C05448=1100.814,341.795,-85.952,179.336,18.021,152.003
C05449=1100.819,342.043,-85.985,179.340,18.025,152.003
C05450=1100.825,342.291,-86.018,179.342,18.028,152.003
C05451=1100.831,342.538,-86.052,179.345,18.031,152.004
C05452=1100.839,342.910,-86.102,179.350,18.036,152.004
C05453=1100.848,343.283,-86.153,179.355,18.040,152.004
C05454=1100.856,343.656,-86.204,179.360,18.045,152.004
C05455=1100.865,344.027,-86.255,179.364,18.049,152.004
C05456=1100.870,344.275,-86.288,179.368,18.053,152.005
C05457=1100.876,344.523,-86.321,179.371,18.056,152.005
C05458=1100.882,344.770,-86.355,179.374,18.059,152.005
C05459=1100.887,345.018,-86.389,179.377,18.062,152.005
C05460=1100.893,345.265,-86.423,179.380,18.065,152.005
C05461=1100.899,345.514,-86.456,179.384,18.069,152.005
C05462=1100.905,345.761,-86.490,179.386,18.072,152.006
C05463=1100.911,346.009,-86.524,179.389,18.075,152.006
C05464=1100.916,346.256,-86.558,179.393,18.078,152.006
C05465=1100.922,346.503,-86.592,179.395,18.082,152.006
C05466=1100.927,346.752,-86.626,179.399,18.085,152.006
C05467=1100.933,346.999,-86.660,179.402,18.088,152.006
C05468=1100.939,347.247,-86.693,179.405,18.091,152.007
C05469=1100.944,347.494,-86.727,179.408,18.095,152.007
C05470=1100.950,347.741,-86.761,179.411,18.098,152.007
C05471=1100.956,347.989,-86.795,179.415,18.101,152.007
C05472=1100.961,348.237,-86.829,179.417,18.104,152.008
C05473=1100.967,348.485,-86.864,179.421,18.108,152.008
C05474=1100.973,348.733,-86.897,179.424,18.111,152.008
C05475=1100.979,348.980,-86.931,179.426,18.114,152.008
C05476=1100.985,349.227,-86.965,179.430,18.118,152.008
C05477=1100.990,349.475,-87.000,179.433,18.121,152.009
C05478=1100.995,349.723,-87.033,179.436,18.125,152.009
C05479=1101.001,349.970,-87.067,179.439,18.128,152.009
C05480=1101.008,350.218,-87.102,179.443,18.132,152.009
C05481=1101.013,350.466,-87.136,179.445,18.135,152.010
C05482=1101.019,350.713,-87.170,179.449,18.138,152.010
C05483=1101.024,350.961,-87.204,179.452,18.142,152.010
C05484=1101.029,351.209,-87.238,179.454,18.145,152.010
C05485=1101.035,351.456,-87.272,179.458,18.149,152.010
C05486=1101.042,351.704,-87.307,179.461,18.151,152.011
C05487=1101.047,351.951,-87.341,179.464,18.155,152.011
C05488=1101.053,352.199,-87.375,179.467,18.159,152.011
C05489=1101.059,352.446,-87.410,179.470,18.162,152.011
C05490=1101.064,352.694,-87.445,179.473,18.166,152.012
C05491=1101.070,352.942,-87.479,179.477,18.169,152.012
C05492=1101.076,353.189,-87.513,179.479,18.172,152.012
C05493=1101.081,353.436,-87.547,179.483,18.176,152.012
C05494=1101.087,353.684,-87.581,179.485,18.179,152.013
C05495=1101.093,353.932,-87.616,179.489,18.183,152.013
C05496=1101.099,354.179,-87.650,179.491,18.187,152.013
C05497=1101.104,354.427,-87.684,179.495,18.190,152.014
C05498=1101.109,354.674,-87.719,179.497,18.194,152.014
C05499=1101.116,354.922,-87.754,179.501,18.197,152.014
C05500=1101.121,355.170,-87.788,179.504,18.201,152.014
C05501=1101.127,355.417,-87.822,179.507,18.205,152.015
C05502=1101.132,355.664,-87.858,179.509,18.208,152.015
C05503=1101.139,355.912,-87.892,179.513,18.212,152.015
C05504=1101.147,356.286,-87.944,179.518,18.218,152.016
C05505=1101.156,356.660,-87.996,179.522,18.223,152.016
C05506=1101.164,357.035,-88.049,179.526,18.228,152.017
C05507=1101.172,357.410,-88.101,179.531,18.234,152.017
C05508=1101.179,357.657,-88.137,179.534,18.238,152.017
C05509=1101.184,357.905,-88.171,179.537,18.241,152.018
C05510=1101.190,358.152,-88.205,179.540,18.245,152.018
C05511=1101.196,358.400,-88.241,179.544,18.249,152.018
C05512=1101.202,358.647,-88.275,179.546,18.253,152.019
C05513=1101.207,358.895,-88.310,179.550,18.256,152.019
C05514=1101.213,359.143,-88.345,179.552,18.260,152.019
C05515=1101.219,359.390,-88.379,179.555,18.264,152.020
C05516=1101.224,359.637,-88.414,179.558,18.267,152.020
C05517=1101.231,359.885,-88.449,179.561,18.271,152.021
C05518=1101.236,360.132,-88.484,179.565,18.275,152.021
C05519=1101.241,360.379,-88.519,179.567,18.279,152.021
C05520=1101.248,360.627,-88.554,179.571,18.283,152.022
C05521=1101.253,360.874,-88.589,179.573,18.286,152.022
C05522=1101.258,361.122,-88.624,179.576,18.290,152.022
C05523=1101.264,361.370,-88.659,179.580,18.295,152.023
C05524=1101.270,361.617,-88.693,179.582,18.298,152.023
C05525=1101.276,361.865,-88.729,179.585,18.302,152.023
C05526=1101.281,362.112,-88.764,179.588,18.306,152.024
C05527=1101.287,362.359,-88.799,179.591,18.310,152.024
C05528=1101.293,362.606,-88.834,179.594,18.314,152.025
C05529=1101.299,362.854,-88.869,179.597,18.317,152.025
C05530=1101.305,363.102,-88.905,179.600,18.322,152.025
C05531=1101.310,363.349,-88.939,179.602,18.325,152.026
C05532=1101.316,363.597,-88.975,179.606,18.329,152.026
C05533=1101.322,363.844,-89.010,179.609,18.333,152.027
C05534=1101.327,364.091,-89.045,179.611,18.337,152.027
C05535=1101.333,364.339,-89.080,179.615,18.341,152.027
C05536=1101.339,364.586,-89.116,179.618,18.346,152.028
C05537=1101.345,364.834,-89.151,179.620,18.349,152.028
C05538=1101.350,365.081,-89.186,179.623,18.353,152.029
C05539=1101.356,365.329,-89.221,179.627,18.358,152.029
C05540=1101.362,365.575,-89.256,179.629,18.361,152.030
C05541=1101.368,365.823,-89.292,179.632,18.366,152.030
C05542=1101.373,366.070,-89.328,179.635,18.370,152.030
C05543=1101.379,366.318,-89.363,179.638,18.374,152.031
C05544=1101.384,366.565,-89.398,179.641,18.378,152.031
C05545=1101.390,366.812,-89.433,179.644,18.382,152.032
C05546=1101.396,367.060,-89.469,179.647,18.386,152.032
C05547=1101.401,367.307,-89.504,179.650,18.390,152.033
C05548=1101.407,367.555,-89.540,179.653,18.395,152.033
C05549=1101.413,367.802,-89.576,179.656,18.399,152.034
C05550=1101.419,368.049,-89.611,179.658,18.403,152.034
C05551=1101.424,368.296,-89.647,179.661,18.407,152.035
C05552=1101.430,368.544,-89.682,179.665,18.411,152.035
C05553=1101.436,368.791,-89.718,179.667,18.415,152.036
C05554=1101.442,369.039,-89.753,179.670,18.420,152.036
C05555=1101.446,369.286,-89.789,179.673,18.424,152.037
C05556=1101.456,369.675,-89.845,179.677,18.431,152.037
C05557=1101.465,370.065,-89.902,179.682,18.438,152.038
C05558=1101.474,370.455,-89.957,179.686,18.444,152.039
C05559=1101.483,370.844,-90.013,179.691,18.451,152.040
C05560=1101.489,371.092,-90.049,179.693,18.455,152.040
C05561=1101.494,371.339,-90.085,179.697,18.459,152.041
C05562=1101.500,371.586,-90.122,179.700,18.464,152.041
C05563=1101.506,371.833,-90.157,179.703,18.469,152.042
C05564=1101.512,372.081,-90.193,179.705,18.472,152.042
C05565=1101.518,372.328,-90.228,179.708,18.477,152.043
C05566=1101.523,372.575,-90.264,179.711,18.482,152.043
C05567=1101.530,372.822,-90.300,179.714,18.486,152.044
C05568=1101.534,373.069,-90.336,179.717,18.491,152.045
C05569=1101.540,373.317,-90.372,179.719,18.495,152.045
C05570=1101.547,373.564,-90.408,179.722,18.499,152.046
C05571=1101.552,373.811,-90.444,179.725,18.503,152.046
C05572=1101.558,374.059,-90.479,179.728,18.508,152.047
C05573=1101.564,374.306,-90.516,179.730,18.512,152.047
C05574=1101.569,374.553,-90.552,179.733,18.517,152.048
C05575=1101.575,374.800,-90.588,179.736,18.521,152.048
C05576=1101.581,375.048,-90.625,179.739,18.526,152.049
C05577=1101.586,375.295,-90.660,179.742,18.531,152.050
C05578=1101.592,375.542,-90.696,179.745,18.535,152.050
C05579=1101.597,375.790,-90.732,179.747,18.540,152.051
C05580=1101.603,376.037,-90.769,179.750,18.545,152.052
C05581=1101.610,376.284,-90.805,179.753,18.549,152.052
C05582=1101.615,376.531,-90.841,179.756,18.554,152.053
C05583=1101.621,376.779,-90.877,179.759,18.559,152.053
C05584=1101.626,377.026,-90.914,179.762,18.564,152.054
C05585=1101.632,377.273,-90.949,179.765,18.568,152.055
C05586=1101.638,377.520,-90.986,179.767,18.572,152.055
C05587=1101.643,377.767,-91.023,179.769,18.577,152.056
C05588=1101.649,378.014,-91.058,179.772,18.582,152.057
C05589=1101.655,378.262,-91.095,179.775,18.587,152.057
C05590=1101.661,378.509,-91.131,179.778,18.592,152.058
C05591=1101.666,378.757,-91.168,179.781,18.596,152.058
C05592=1101.672,379.003,-91.204,179.784,18.601,152.059
C05593=1101.677,379.251,-91.240,179.787,18.606,152.060
C05594=1101.684,379.498,-91.277,179.789,18.610,152.060
C05595=1101.689,379.746,-91.314,179.792,18.615,152.061
C05596=1101.695,379.992,-91.350,179.794,18.620,152.062
C05597=1101.700,380.240,-91.386,179.797,18.625,152.062
C05598=1101.706,380.487,-91.423,179.800,18.630,152.063
C05599=1101.712,380.734,-91.460,179.803,18.635,152.064
C05600=1101.718,380.981,-91.496,179.806,18.640,152.064
C05601=1101.723,381.228,-91.533,179.808,18.645,152.065
C05602=1101.729,381.476,-91.569,179.811,18.650,152.066
C05603=1101.735,381.723,-91.606,179.814,18.655,152.067
C05604=1101.741,381.970,-91.642,179.817,18.659,152.067
C05605=1101.746,382.217,-91.679,179.819,18.664,152.068
C05606=1101.753,382.464,-91.715,179.822,18.669,152.069
C05607=1101.758,382.711,-91.752,179.824,18.674,152.069
C05608=1101.768,383.128,-91.814,179.829,18.683,152.071
C05609=1101.777,383.543,-91.876,179.833,18.691,152.072
C05610=1101.787,383.960,-91.938,179.838,18.700,152.073
C05611=1101.796,384.376,-92.000,179.843,18.708,152.074
C05612=1101.802,384.624,-92.037,179.845,18.714,152.075
C05613=1101.808,384.871,-92.073,179.848,18.719,152.076
C05614=1101.814,385.118,-92.111,179.850,18.724,152.077
C05615=1101.820,385.366,-92.148,179.853,18.729,152.078
C05616=1101.825,385.612,-92.185,179.856,18.734,152.078
C05617=1101.831,385.859,-92.221,179.858,18.739,152.079
C05618=1101.837,386.106,-92.258,179.861,18.745,152.080
C05619=1101.842,386.353,-92.295,179.864,18.750,152.081
C05620=1101.848,386.601,-92.333,179.866,18.755,152.082
C05621=1101.854,386.848,-92.370,179.869,18.760,152.082
C05622=1101.860,387.095,-92.407,179.871,18.766,152.083
C05623=1101.865,387.341,-92.443,179.874,18.771,152.084
C05624=1101.871,387.589,-92.480,179.877,18.777,152.085
C05625=1101.876,387.836,-92.517,179.880,18.782,152.086
C05626=1101.882,388.083,-92.555,179.882,18.787,152.087
C05627=1101.888,388.330,-92.592,179.885,18.793,152.087
C05628=1101.894,388.577,-92.629,179.888,18.798,152.088
C05629=1101.900,388.824,-92.666,179.890,18.803,152.089
C05630=1101.906,389.071,-92.703,179.893,18.809,152.090
C05631=1101.911,389.319,-92.741,179.895,18.814,152.091
C05632=1101.917,389.565,-92.778,179.898,18.820,152.092
C05633=1101.923,389.813,-92.815,179.900,18.825,152.092
C05634=1101.929,390.059,-92.853,179.903,18.830,152.093
C05635=1101.934,390.307,-92.890,179.906,18.836,152.094
C05636=1101.940,390.554,-92.928,179.909,18.842,152.095
C05637=1101.947,390.801,-92.964,179.911,18.847,152.096
C05638=1101.953,391.047,-93.002,179.913,18.852,152.097
C05639=1101.958,391.295,-93.039,179.916,18.858,152.098
C05640=1101.964,391.541,-93.077,179.918,18.863,152.099
C05641=1101.970,391.789,-93.114,179.921,18.869,152.100
C05642=1101.976,392.036,-93.152,179.923,18.875,152.101
C05643=1101.981,392.283,-93.189,179.926,18.881,152.101
C05644=1101.987,392.530,-93.226,179.929,18.886,152.102
C05645=1101.993,392.777,-93.264,179.931,18.892,152.103
C05646=1101.999,393.024,-93.301,179.934,18.897,152.104
C05647=1102.004,393.271,-93.340,179.936,18.903,152.105
C05648=1102.009,393.518,-93.377,179.938,18.909,152.106
C05649=1102.015,393.765,-93.414,179.942,18.915,152.107
C05650=1102.021,394.012,-93.452,179.944,18.921,152.108
C05651=1102.027,394.259,-93.489,179.946,18.926,152.109
C05652=1102.033,394.507,-93.527,179.949,18.932,152.110
C05653=1102.039,394.753,-93.565,179.951,18.938,152.111
C05654=1102.044,395.000,-93.603,179.953,18.943,152.112
C05655=1102.050,395.248,-93.640,179.956,18.950,152.113
C05656=1102.056,395.494,-93.678,179.959,18.955,152.114
C05657=1102.062,395.741,-93.716,179.961,18.961,152.115
C05658=1102.068,395.988,-93.754,179.963,18.967,152.116
C05659=1102.072,396.236,-93.791,179.966,18.973,152.117
C05660=1102.078,396.450,-93.824,179.968,18.978,152.118
C05661=1102.083,396.665,-93.857,179.970,18.984,152.119
C05662=1102.088,396.878,-93.890,179.972,18.989,152.120
C05663=1102.093,397.093,-93.924,179.975,18.994,152.121
C05664=1102.098,397.307,-93.955,179.976,18.999,152.121
C05665=1102.103,397.521,-93.989,179.979,19.004,152.122
C05666=1102.108,397.737,-94.022,179.980,19.010,152.123
C05667=1102.113,397.950,-94.055,179.983,19.015,152.124
C05668=1102.118,398.197,-94.093,179.985,19.021,152.125
C05669=1102.125,398.445,-94.131,179.988,19.027,152.126
C05670=1102.131,398.691,-94.169,179.990,19.033,152.128
C05671=1102.136,398.938,-94.207,179.992,19.039,152.129
C05672=1102.142,399.185,-94.245,179.995,19.045,152.130
C05673=1102.148,399.432,-94.283,179.998,19.052,152.131
C05674=1102.153,399.680,-94.321,180.000,19.058,152.132
C05675=1102.159,399.926,-94.359,-179.998,19.064,152.133
C05676=1102.164,400.173,-94.398,-179.995,19.070,152.134
C05677=1102.171,400.421,-94.436,-179.993,19.077,152.135
C05678=1102.176,400.668,-94.474,-179.991,19.083,152.136
C05679=1102.182,400.915,-94.512,-179.988,19.089,152.137
C05680=1102.188,401.161,-94.550,-179.986,19.096,152.139
C05681=1102.194,401.408,-94.589,-179.984,19.102,152.140
C05682=1102.199,401.656,-94.627,-179.981,19.109,152.141
C05683=1102.205,401.902,-94.665,-179.979,19.115,152.142
C05684=1102.210,402.149,-94.703,-179.976,19.122,152.143
C05685=1102.217,402.396,-94.742,-179.974,19.128,152.144
C05686=1102.222,402.643,-94.781,-179.972,19.134,152.146
C05687=1102.228,402.890,-94.818,-179.969,19.141,152.147
C05688=1102.234,403.138,-94.857,-179.967,19.147,152.148
C05689=1102.240,403.384,-94.896,-179.964,19.154,152.149
C05690=1102.245,403.631,-94.934,-179.962,19.160,152.150
C05691=1102.252,403.878,-94.972,-179.960,19.167,152.152
C05692=1102.257,404.125,-95.011,-179.958,19.173,152.153
C05693=1102.262,404.372,-95.049,-179.956,19.180,152.154
C05694=1102.269,404.619,-95.088,-179.953,19.187,152.155
C05695=1102.274,404.866,-95.127,-179.951,19.193,152.156
C05696=1102.279,405.113,-95.165,-179.948,19.200,152.158
C05697=1102.286,405.360,-95.204,-179.946,19.206,152.159
C05698=1102.291,405.607,-95.242,-179.944,19.214,152.160
C05699=1102.297,405.854,-95.282,-179.942,19.220,152.162
C05700=1102.303,406.101,-95.319,-179.939,19.227,152.163
C05701=1102.309,406.347,-95.358,-179.937,19.234,152.164
C05702=1102.315,406.595,-95.397,-179.935,19.241,152.165
C05703=1102.320,406.841,-95.436,-179.932,19.247,152.167
C05704=1102.327,407.089,-95.474,-179.930,19.254,152.168
C05705=1102.332,407.335,-95.513,-179.927,19.262,152.169
C05706=1102.337,407.582,-95.552,-179.925,19.268,152.171
C05707=1102.343,407.829,-95.591,-179.923,19.275,152.172
C05708=1102.349,408.076,-95.630,-179.921,19.282,152.173
C05709=1102.355,408.323,-95.668,-179.918,19.289,152.175
C05710=1102.361,408.570,-95.707,-179.917,19.296,152.176
C05711=1102.367,408.817,-95.747,-179.914,19.303,152.177
C05712=1102.372,409.064,-95.785,-179.912,19.311,152.179
C05713=1102.377,409.310,-95.824,-179.910,19.317,152.180
C05714=1102.384,409.557,-95.864,-179.907,19.325,152.181
C05715=1102.389,409.804,-95.903,-179.905,19.332,152.183
C05716=1102.394,410.018,-95.936,-179.903,19.338,152.184
C05717=1102.399,410.233,-95.970,-179.902,19.344,152.185
C05718=1102.404,410.447,-96.004,-179.900,19.351,152.186
C05719=1102.409,410.661,-96.038,-179.898,19.357,152.188
C05720=1102.414,410.876,-96.072,-179.896,19.363,152.189
C05721=1102.419,411.090,-96.106,-179.894,19.370,152.190
C05722=1102.424,411.304,-96.140,-179.892,19.376,152.191
C05723=1102.429,411.519,-96.174,-179.890,19.382,152.193
C05724=1102.435,411.766,-96.213,-179.887,19.390,152.194
C05725=1102.441,412.012,-96.252,-179.886,19.397,152.196
C05726=1102.447,412.259,-96.292,-179.883,19.405,152.197
C05727=1102.452,412.506,-96.331,-179.881,19.412,152.198
C05728=1102.458,412.753,-96.370,-179.878,19.419,152.200
C05729=1102.464,412.999,-96.409,-179.877,19.426,152.201
C05730=1102.470,413.247,-96.449,-179.874,19.434,152.203
C05731=1102.476,413.494,-96.488,-179.872,19.442,152.204
C05732=1102.481,413.740,-96.527,-179.870,19.450,152.206
C05733=1102.487,413.988,-96.567,-179.868,19.457,152.207
C05734=1102.492,414.234,-96.606,-179.866,19.464,152.209
C05735=1102.498,414.481,-96.646,-179.863,19.472,152.210
C05736=1102.505,414.728,-96.686,-179.861,19.480,152.212
C05737=1102.510,414.974,-96.725,-179.859,19.487,152.213
C05738=1102.516,415.221,-96.764,-179.857,19.495,152.215
C05739=1102.522,415.468,-96.803,-179.855,19.502,152.216
C05740=1102.528,415.715,-96.843,-179.853,19.510,152.218
C05741=1102.534,415.961,-96.883,-179.850,19.518,152.220
C05742=1102.540,416.208,-96.922,-179.848,19.526,152.221
C05743=1102.546,416.455,-96.961,-179.846,19.534,152.223
C05744=1102.551,416.702,-97.001,-179.844,19.541,152.224
C05745=1102.557,416.948,-97.041,-179.842,19.549,152.226
C05746=1102.563,417.195,-97.081,-179.840,19.557,152.227
C05747=1102.569,417.442,-97.120,-179.838,19.565,152.229
C05748=1102.574,417.689,-97.160,-179.836,19.573,152.231
C05749=1102.580,417.936,-97.200,-179.833,19.581,152.232
C05750=1102.586,418.183,-97.239,-179.831,19.590,152.234
C05751=1102.591,418.429,-97.280,-179.829,19.598,152.236
C05752=1102.597,418.676,-97.319,-179.827,19.606,152.237
C05753=1102.603,418.922,-97.359,-179.825,19.614,152.239
C05754=1102.608,419.169,-97.399,-179.823,19.622,152.241
C05755=1102.615,419.416,-97.439,-179.821,19.630,152.242
C05756=1102.621,419.663,-97.478,-179.819,19.638,152.244
C05757=1102.626,419.909,-97.519,-179.817,19.647,152.246
C05758=1102.632,420.156,-97.558,-179.815,19.655,152.247
C05759=1102.638,420.403,-97.598,-179.813,19.664,152.249
C05760=1102.643,420.649,-97.639,-179.810,19.671,152.251
C05761=1102.649,420.896,-97.678,-179.808,19.680,152.253
C05762=1102.655,421.143,-97.719,-179.806,19.688,152.254
C05763=1102.661,421.390,-97.758,-179.804,19.697,152.256
C05764=1102.667,421.636,-97.798,-179.802,19.705,152.258
C05765=1102.673,421.883,-97.839,-179.800,19.713,152.260
C05766=1102.679,422.129,-97.879,-179.799,19.722,152.261
C05767=1102.684,422.377,-97.919,-179.797,19.731,152.263
C05768=1102.691,422.623,-97.959,-179.795,19.739,152.265
C05769=1102.696,422.869,-98.000,-179.793,19.747,152.267
C05770=1102.702,423.116,-98.040,-179.791,19.756,152.269
C05771=1102.707,423.363,-98.080,-179.789,19.764,152.270
C05772=1102.713,423.584,-98.116,-179.787,19.773,152.272
C05773=1102.718,423.805,-98.152,-179.785,19.780,152.274
C05774=1102.723,424.026,-98.189,-179.783,19.789,152.275
C05775=1102.728,424.248,-98.225,-179.782,19.796,152.277
C05776=1102.733,424.468,-98.260,-179.780,19.804,152.279
C05777=1102.738,424.689,-98.297,-179.778,19.812,152.280
C05778=1102.744,424.910,-98.333,-179.776,19.820,152.282
C05779=1102.749,425.132,-98.369,-179.775,19.828,152.284
C05780=1102.755,425.378,-98.409,-179.772,19.837,152.286
C05781=1102.760,425.625,-98.450,-179.771,19.846,152.288
C05782=1102.766,425.871,-98.491,-179.769,19.855,152.290
C05783=1102.772,426.118,-98.531,-179.767,19.863,152.291
C05784=1102.778,426.365,-98.571,-179.765,19.873,152.294
C05785=1102.784,426.611,-98.613,-179.763,19.882,152.295
C05786=1102.790,426.857,-98.653,-179.761,19.891,152.297
C05787=1102.795,427.104,-98.693,-179.759,19.900,152.299
C05788=1102.801,427.350,-98.734,-179.758,19.909,152.301
C05789=1102.807,427.597,-98.774,-179.755,19.919,152.303
C05790=1102.813,427.844,-98.815,-179.754,19.927,152.305
C05791=1102.819,428.091,-98.856,-179.752,19.937,152.307
C05792=1102.825,428.337,-98.897,-179.750,19.946,152.309
C05793=1102.831,428.583,-98.937,-179.748,19.956,152.311
C05794=1102.837,428.830,-98.978,-179.746,19.965,152.313
C05795=1102.842,429.077,-99.019,-179.745,19.974,152.315
C05796=1102.848,429.322,-99.060,-179.742,19.984,152.317
C05797=1102.854,429.569,-99.100,-179.741,19.993,152.320
C05798=1102.860,429.816,-99.141,-179.739,20.002,152.322
C05799=1102.866,430.062,-99.182,-179.737,20.012,152.324
C05800=1102.871,430.309,-99.223,-179.735,20.022,152.326
C05801=1102.877,430.555,-99.265,-179.734,20.031,152.328
C05802=1102.883,430.802,-99.305,-179.732,20.041,152.330
C05803=1102.889,431.049,-99.346,-179.730,20.050,152.332
C05804=1102.894,431.295,-99.388,-179.729,20.060,152.334
C05805=1102.900,431.542,-99.428,-179.727,20.070,152.337
C05806=1102.906,431.788,-99.470,-179.725,20.080,152.339
C05807=1102.912,432.035,-99.510,-179.723,20.090,152.341
C05808=1102.918,432.281,-99.551,-179.722,20.099,152.343
C05809=1102.924,432.527,-99.593,-179.720,20.109,152.345
C05810=1102.930,432.774,-99.634,-179.718,20.119,152.348
C05811=1102.936,433.020,-99.675,-179.717,20.129,152.350
C05812=1102.942,433.267,-99.716,-179.715,20.139,152.352
C05813=1102.948,433.513,-99.757,-179.713,20.149,152.354
C05814=1102.953,433.759,-99.799,-179.711,20.159,152.356
C05815=1102.958,434.006,-99.840,-179.710,20.169,152.359
C05816=1102.964,434.252,-99.881,-179.708,20.180,152.361
C05817=1102.970,434.499,-99.923,-179.707,20.190,152.363
C05818=1102.976,434.745,-99.964,-179.705,20.200,152.366
C05819=1102.982,434.992,-100.005,-179.703,20.210,152.368
C05820=1102.988,435.238,-100.047,-179.701,20.221,152.370
C05821=1102.994,435.484,-100.088,-179.700,20.231,152.373
C05822=1102.999,435.731,-100.130,-179.698,20.242,152.375
C05823=1103.005,435.977,-100.172,-179.697,20.251,152.377
C05824=1103.011,436.223,-100.213,-179.695,20.262,152.380
C05825=1103.017,436.469,-100.254,-179.694,20.272,152.382
C05826=1103.022,436.716,-100.295,-179.692,20.283,152.385
C05827=1103.028,436.963,-100.337,-179.690,20.294,152.387
C05828=1103.038,437.358,-100.404,-179.688,20.311,152.391
C05829=1103.047,437.753,-100.471,-179.685,20.328,152.395
C05830=1103.056,438.149,-100.538,-179.684,20.345,152.399
C05831=1103.066,438.544,-100.605,-179.681,20.362,152.403
C05832=1103.072,438.791,-100.647,-179.679,20.374,152.405
C05833=1103.077,439.037,-100.688,-179.678,20.384,152.408
C05834=1103.083,439.283,-100.730,-179.676,20.395,152.410
C05835=1103.089,439.530,-100.772,-179.674,20.406,152.413
C05836=1103.095,439.776,-100.814,-179.674,20.417,152.415
C05837=1103.101,440.022,-100.856,-179.672,20.428,152.418
C05838=1103.107,440.268,-100.897,-179.670,20.439,152.420
C05839=1103.113,440.515,-100.939,-179.669,20.450,152.423
C05840=1103.119,440.761,-100.981,-179.668,20.461,152.426
C05841=1103.125,441.008,-101.024,-179.666,20.473,152.428
C05842=1103.131,441.254,-101.065,-179.664,20.484,152.431
C05843=1103.136,441.500,-101.108,-179.664,20.495,152.433
C05844=1103.142,441.746,-101.150,-179.662,20.507,152.436
C05845=1103.148,441.992,-101.191,-179.661,20.518,152.439
C05846=1103.154,442.239,-101.234,-179.659,20.530,152.442
C05847=1103.160,442.485,-101.276,-179.657,20.541,152.444
C05848=1103.165,442.731,-101.318,-179.657,20.552,152.447
C05849=1103.172,442.977,-101.360,-179.655,20.564,152.450
C05850=1103.177,443.223,-101.402,-179.654,20.576,152.453
C05851=1103.183,443.470,-101.445,-179.652,20.588,152.455
C05852=1103.189,443.716,-101.487,-179.652,20.599,152.458
C05853=1103.194,443.962,-101.529,-179.650,20.611,152.461
C05854=1103.201,444.208,-101.572,-179.650,20.622,152.464
C05855=1103.206,444.455,-101.614,-179.649,20.635,152.466
C05856=1103.212,444.701,-101.657,-179.648,20.646,152.469
C05857=1103.218,444.947,-101.698,-179.648,20.658,152.472
C05858=1103.224,445.194,-101.741,-179.647,20.669,152.475
C05859=1103.230,445.439,-101.784,-179.648,20.680,152.478
C05860=1103.235,445.686,-101.826,-179.647,20.692,152.481
C05861=1103.242,445.932,-101.869,-179.648,20.703,152.484
C05862=1103.248,446.178,-101.911,-179.647,20.715,152.487
C05863=1103.253,446.424,-101.953,-179.648,20.727,152.490
C05864=1103.259,446.671,-101.996,-179.648,20.738,152.493
C05865=1103.265,446.917,-102.039,-179.649,20.749,152.496
C05866=1103.270,447.163,-102.082,-179.650,20.761,152.499
C05867=1103.277,447.410,-102.123,-179.650,20.772,152.502
C05868=1103.282,447.656,-102.166,-179.651,20.784,152.505
C05869=1103.288,447.901,-102.209,-179.652,20.795,152.508
C05870=1103.294,448.148,-102.252,-179.653,20.807,152.511
C05871=1103.300,448.394,-102.294,-179.654,20.818,152.514
C05872=1103.306,448.641,-102.337,-179.655,20.830,152.517
C05873=1103.312,448.887,-102.379,-179.657,20.841,152.521
C05874=1103.317,449.133,-102.422,-179.658,20.852,152.524
C05875=1103.323,449.379,-102.465,-179.660,20.864,152.527
C05876=1103.329,449.625,-102.508,-179.662,20.875,152.530
C05877=1103.336,449.871,-102.551,-179.663,20.886,152.533
C05878=1103.341,450.117,-102.593,-179.665,20.898,152.536
C05879=1103.347,450.364,-102.637,-179.667,20.909,152.539
C05880=1102.945,450.357,-102.771,-179.739,21.135,152.609
C05881=1102.939,450.111,-102.728,-179.737,21.124,152.606
C05882=1102.933,449.864,-102.685,-179.736,21.112,152.603
C05883=1102.928,449.618,-102.642,-179.734,21.101,152.599
C05884=1102.921,449.372,-102.600,-179.732,21.090,152.596
C05885=1102.915,449.126,-102.557,-179.731,21.078,152.593
C05886=1102.910,448.880,-102.514,-179.729,21.067,152.590
C05887=1102.904,448.633,-102.471,-179.728,21.055,152.587
C05888=1102.898,448.388,-102.428,-179.727,21.044,152.584
C05889=1102.892,448.141,-102.385,-179.725,21.033,152.581
C05890=1102.886,447.895,-102.343,-179.725,21.021,152.577
C05891=1102.880,447.648,-102.301,-179.723,21.010,152.574
C05892=1102.874,447.402,-102.258,-179.723,20.998,152.571
C05893=1102.869,447.156,-102.215,-179.722,20.986,152.568
C05894=1102.863,446.910,-102.172,-179.722,20.974,152.565
C05895=1102.857,446.664,-102.130,-179.721,20.963,152.562
C05896=1102.851,446.418,-102.087,-179.721,20.951,152.559
C05897=1102.845,446.171,-102.045,-179.720,20.940,152.556
C05898=1102.840,445.925,-102.002,-179.721,20.928,152.553
C05899=1102.833,445.679,-101.959,-179.720,20.917,152.550
C05900=1102.827,445.433,-101.916,-179.721,20.905,152.547
C05901=1102.822,445.187,-101.874,-179.721,20.893,152.544
C05902=1102.815,444.940,-101.832,-179.721,20.882,152.541
C05903=1102.810,444.694,-101.789,-179.721,20.870,152.539
C05904=1102.805,444.448,-101.747,-179.723,20.858,152.536
C05905=1102.798,444.202,-101.705,-179.723,20.846,152.533
C05906=1102.792,443.956,-101.662,-179.724,20.835,152.530
C05907=1102.787,443.709,-101.620,-179.725,20.823,152.527
C05908=1102.781,443.464,-101.578,-179.727,20.811,152.524
C05909=1102.775,443.217,-101.534,-179.727,20.800,152.522
C05910=1102.769,442.971,-101.493,-179.729,20.788,152.519
C05911=1102.763,442.725,-101.450,-179.730,20.776,152.516
C05912=1102.757,442.478,-101.408,-179.732,20.764,152.513
C05913=1102.751,442.232,-101.366,-179.734,20.753,152.511
C05914=1102.745,441.986,-101.324,-179.734,20.741,152.508
C05915=1102.740,441.740,-101.281,-179.736,20.730,152.505
C05916=1102.734,441.494,-101.240,-179.738,20.718,152.503
C05917=1102.728,441.247,-101.197,-179.739,20.706,152.500
C05918=1102.722,441.001,-101.155,-179.740,20.696,152.497
C05919=1102.716,440.754,-101.113,-179.742,20.684,152.495
C05920=1102.710,440.509,-101.071,-179.744,20.673,152.492
C05921=1102.704,440.262,-101.029,-179.745,20.662,152.489
C05922=1102.698,440.015,-100.987,-179.746,20.650,152.487
C05923=1102.692,439.769,-100.946,-179.748,20.639,152.484
C05924=1102.686,439.524,-100.904,-179.750,20.628,152.482
C05925=1102.681,439.277,-100.862,-179.751,20.618,152.479
C05926=1102.674,439.030,-100.820,-179.753,20.606,152.477
C05927=1102.668,438.784,-100.778,-179.754,20.595,152.474
C05928=1102.663,438.538,-100.735,-179.755,20.584,152.471
C05929=1102.654,438.148,-100.670,-179.758,20.567,152.468
C05930=1102.645,437.759,-100.604,-179.760,20.550,152.464
C05931=1102.635,437.369,-100.538,-179.763,20.533,152.460
C05932=1102.626,436.980,-100.472,-179.765,20.516,152.456
C05933=1102.620,436.733,-100.430,-179.767,20.505,152.454
C05934=1102.614,436.486,-100.388,-179.769,20.495,152.451
C05935=1102.608,436.240,-100.347,-179.770,20.484,152.449
C05936=1102.602,435.994,-100.305,-179.772,20.473,152.446
C05937=1102.596,435.748,-100.264,-179.774,20.463,152.444
C05938=1102.591,435.501,-100.222,-179.776,20.452,152.442
C05939=1102.585,435.255,-100.181,-179.777,20.442,152.439
C05940=1102.579,435.008,-100.140,-179.779,20.432,152.437
C05941=1102.573,434.762,-100.098,-179.780,20.422,152.435
C05942=1102.567,434.516,-100.057,-179.782,20.411,152.432
C05943=1102.561,434.270,-100.015,-179.783,20.401,152.430
C05944=1102.556,434.023,-99.973,-179.786,20.390,152.428
C05945=1102.551,433.776,-99.933,-179.787,20.380,152.425
C05946=1102.545,433.530,-99.891,-179.789,20.370,152.423
C05947=1102.539,433.284,-99.850,-179.790,20.360,152.421
C05948=1102.533,433.037,-99.809,-179.793,20.350,152.418
C05949=1102.527,432.791,-99.767,-179.794,20.340,152.416
C05950=1102.521,432.545,-99.726,-179.796,20.330,152.414
C05951=1102.515,432.298,-99.685,-179.798,20.320,152.412
C05952=1102.509,432.052,-99.644,-179.800,20.310,152.410
C05953=1102.504,431.806,-99.602,-179.801,20.300,152.407
C05954=1102.498,431.559,-99.562,-179.803,20.290,152.405
C05955=1102.492,431.312,-99.520,-179.805,20.280,152.403
C05956=1102.486,431.066,-99.479,-179.807,20.271,152.401
C05957=1102.480,430.819,-99.438,-179.809,20.261,152.399
C05958=1102.474,430.573,-99.398,-179.810,20.251,152.397
C05959=1102.468,430.327,-99.356,-179.812,20.242,152.394
C05960=1102.462,430.080,-99.316,-179.814,20.232,152.392
C05961=1102.457,429.833,-99.275,-179.816,20.222,152.390
C05962=1102.451,429.587,-99.233,-179.817,20.213,152.388
C05963=1102.445,429.340,-99.193,-179.820,20.203,152.386
C05964=1102.439,429.094,-99.151,-179.821,20.194,152.384
C05965=1102.434,428.847,-99.110,-179.823,20.184,152.382
C05966=1102.427,428.601,-99.070,-179.825,20.175,152.380
C05967=1102.422,428.354,-99.030,-179.827,20.165,152.378
C05968=1102.416,428.107,-98.988,-179.829,20.156,152.376
C05969=1102.411,427.861,-98.948,-179.830,20.147,152.374
C05970=1102.404,427.615,-98.908,-179.833,20.137,152.372
C05971=1102.399,427.368,-98.867,-179.834,20.128,152.370
C05972=1102.393,427.122,-98.825,-179.836,20.119,152.368
C05973=1102.386,426.875,-98.785,-179.838,20.110,152.366
C05974=1102.381,426.628,-98.744,-179.841,20.100,152.364
C05975=1102.375,426.382,-98.704,-179.842,20.092,152.362
C05976=1102.369,426.135,-98.664,-179.844,20.082,152.360
C05977=1102.363,425.888,-98.623,-179.846,20.073,152.358
C05978=1102.358,425.642,-98.582,-179.848,20.064,152.356
C05979=1102.351,425.396,-98.542,-179.850,20.055,152.354
C05980=1102.346,425.149,-98.502,-179.852,20.046,152.352
C05981=1102.341,424.928,-98.465,-179.854,20.038,152.350
C05982=1102.335,424.707,-98.429,-179.856,20.030,152.349
C05983=1102.330,424.485,-98.393,-179.858,20.022,152.347
C05984=1102.325,424.263,-98.356,-179.859,20.014,152.345
C05985=1102.319,424.042,-98.320,-179.861,20.006,152.344
C05986=1102.315,423.821,-98.284,-179.863,19.999,152.342
C05987=1102.310,423.599,-98.247,-179.865,19.990,152.340
C05988=1102.304,423.378,-98.211,-179.866,19.982,152.338
C05989=1102.299,423.132,-98.170,-179.868,19.974,152.337
C05990=1102.293,422.885,-98.131,-179.870,19.965,152.335
C05991=1102.287,422.638,-98.090,-179.873,19.956,152.333
C05992=1102.281,422.392,-98.050,-179.875,19.948,152.331
C05993=1102.275,422.145,-98.009,-179.877,19.939,152.330
C05994=1102.269,421.899,-97.970,-179.879,19.930,152.328
C05995=1102.264,421.652,-97.929,-179.881,19.922,152.326
C05996=1102.258,421.405,-97.889,-179.883,19.914,152.324
C05997=1102.251,421.159,-97.849,-179.885,19.905,152.322
C05998=1102.246,420.911,-97.809,-179.887,19.897,152.321
C05999=1102.240,420.665,-97.769,-179.889,19.888,152.319
C06000=1102.234,420.419,-97.729,-179.891,19.880,152.317
C06001=1102.228,420.171,-97.689,-179.893,19.872,152.315
C06002=1102.222,419.925,-97.649,-179.895,19.863,152.314
C06003=1102.217,419.678,-97.609,-179.897,19.855,152.312
C06004=1102.211,419.432,-97.569,-179.899,19.847,152.310
C06005=1102.204,419.185,-97.529,-179.901,19.838,152.309
C06006=1102.200,418.938,-97.489,-179.903,19.830,152.307
C06007=1102.193,418.692,-97.449,-179.906,19.822,152.305
C06008=1102.187,418.445,-97.410,-179.908,19.814,152.303
C06009=1102.182,418.199,-97.370,-179.910,19.805,152.302
C06010=1102.176,417.951,-97.330,-179.912,19.797,152.300
C06011=1102.170,417.704,-97.291,-179.914,19.789,152.299
C06012=1102.165,417.458,-97.250,-179.916,19.781,152.297
C06013=1102.159,417.211,-97.211,-179.919,19.773,152.295
C06014=1102.153,416.965,-97.171,-179.920,19.766,152.294
C06015=1102.148,416.718,-97.131,-179.922,19.757,152.292
C06016=1102.142,416.471,-97.092,-179.924,19.749,152.290
C06017=1102.135,416.224,-97.051,-179.927,19.742,152.289
C06018=1102.130,415.978,-97.012,-179.929,19.734,152.287
C06019=1102.124,415.731,-96.973,-179.931,19.726,152.286
C06020=1102.118,415.483,-96.934,-179.934,19.718,152.284
C06021=1102.112,415.238,-96.894,-179.936,19.710,152.282
C06022=1102.107,414.990,-96.854,-179.938,19.703,152.281
C06023=1102.101,414.743,-96.814,-179.940,19.695,152.279
C06024=1102.095,414.497,-96.775,-179.942,19.687,152.278
C06025=1102.089,414.249,-96.736,-179.945,19.679,152.276
C06026=1102.083,414.003,-96.696,-179.947,19.672,152.275
C06027=1102.077,413.757,-96.657,-179.949,19.664,152.273
C06028=1102.071,413.509,-96.617,-179.951,19.657,152.272
C06029=1102.066,413.263,-96.578,-179.953,19.649,152.270
C06030=1102.060,413.016,-96.539,-179.956,19.641,152.269
C06031=1102.053,412.769,-96.499,-179.957,19.634,152.267
C06032=1102.048,412.522,-96.460,-179.960,19.627,152.266
C06033=1102.042,412.275,-96.421,-179.962,19.619,152.264
C06034=1102.036,412.029,-96.382,-179.965,19.611,152.263
C06035=1102.030,411.782,-96.342,-179.966,19.604,152.261
C06036=1102.025,411.535,-96.303,-179.969,19.597,152.260
C06037=1102.020,411.321,-96.270,-179.971,19.590,152.259
C06038=1102.015,411.105,-96.235,-179.973,19.584,152.257
C06039=1102.010,410.891,-96.201,-179.975,19.578,152.256
C06040=1102.005,410.677,-96.167,-179.977,19.571,152.255
C06041=1102.000,410.462,-96.133,-179.979,19.565,152.254
C06042=1101.995,410.247,-96.099,-179.981,19.558,152.252
C06043=1101.989,410.033,-96.065,-179.983,19.552,152.251
C06044=1101.985,409.818,-96.030,-179.985,19.545,152.250
C06045=1101.979,409.571,-95.993,-179.987,19.539,152.249
C06046=1101.973,409.324,-95.953,-179.989,19.531,152.247
C06047=1101.968,409.078,-95.914,-179.992,19.524,152.246
C06048=1101.962,408.831,-95.875,-179.993,19.517,152.244
C06049=1101.956,408.584,-95.836,-179.996,19.510,152.243
C06050=1101.950,408.336,-95.797,-179.998,19.503,152.242
C06051=1101.945,408.090,-95.758,180.000,19.496,152.240
C06052=1101.939,407.844,-95.719,179.997,19.488,152.239
C06053=1101.934,407.596,-95.680,179.995,19.482,152.238
C06054=1101.927,407.350,-95.642,179.993,19.474,152.236
C06055=1101.922,407.102,-95.603,179.991,19.468,152.235
C06056=1101.916,406.855,-95.564,179.988,19.460,152.234
C06057=1101.910,406.608,-95.524,179.986,19.454,152.232
C06058=1101.904,406.362,-95.487,179.984,19.447,152.231
C06059=1101.899,406.115,-95.448,179.982,19.440,152.230
C06060=1101.893,405.867,-95.409,179.979,19.433,152.229
C06061=1101.887,405.621,-95.370,179.977,19.427,152.227
C06062=1101.881,405.374,-95.332,179.974,19.419,152.226
C06063=1101.876,405.127,-95.293,179.972,19.412,152.225
C06064=1101.870,404.880,-95.254,179.969,19.406,152.224
C06065=1101.864,404.633,-95.215,179.968,19.399,152.222
C06066=1101.858,404.386,-95.177,179.965,19.392,152.221
C06067=1101.853,404.138,-95.138,179.963,19.386,152.220
C06068=1101.846,403.892,-95.100,179.960,19.379,152.219
C06069=1101.841,403.645,-95.061,179.958,19.372,152.217
C06070=1101.834,403.398,-95.023,179.955,19.366,152.216
C06071=1101.829,403.151,-94.984,179.953,19.359,152.215
C06072=1101.824,402.904,-94.946,179.950,19.352,152.214
C06073=1101.817,402.657,-94.907,179.948,19.346,152.212
C06074=1101.812,402.410,-94.869,179.946,19.340,152.211
C06075=1101.806,402.164,-94.831,179.943,19.333,152.210
C06076=1101.800,401.916,-94.792,179.941,19.327,152.209
C06077=1101.794,401.670,-94.754,179.938,19.320,152.208
C06078=1101.789,401.423,-94.715,179.936,19.314,152.207
C06079=1101.783,401.176,-94.678,179.934,19.308,152.205
C06080=1101.777,400.928,-94.639,179.931,19.301,152.204
C06081=1101.771,400.681,-94.601,179.929,19.295,152.203
C06082=1101.766,400.435,-94.562,179.926,19.288,152.202
C06083=1101.760,400.188,-94.524,179.924,19.281,152.201
C06084=1101.754,399.941,-94.486,179.922,19.275,152.200
C06085=1101.748,399.694,-94.448,179.919,19.269,152.199
C06086=1101.743,399.447,-94.410,179.917,19.263,152.197
C06087=1101.737,399.200,-94.372,179.915,19.256,152.196
C06088=1101.731,398.953,-94.334,179.912,19.250,152.195
C06089=1101.726,398.706,-94.295,179.910,19.244,152.194
C06090=1101.720,398.459,-94.258,179.908,19.238,152.193
C06091=1101.714,398.212,-94.220,179.906,19.232,152.192
C06092=1101.708,397.964,-94.181,179.902,19.225,152.191
C06093=1101.703,397.751,-94.148,179.901,19.221,152.190
C06094=1101.698,397.536,-94.116,179.898,19.215,152.189
C06095=1101.693,397.321,-94.082,179.897,19.210,152.188
C06096=1101.688,397.106,-94.049,179.894,19.204,152.187
C06097=1101.683,396.891,-94.017,179.892,19.199,152.186
C06098=1101.678,396.677,-93.983,179.890,19.194,152.185
C06099=1101.673,396.463,-93.951,179.887,19.188,152.184
C06100=1101.668,396.248,-93.918,179.886,19.184,152.184
C06101=1101.662,396.001,-93.880,179.883,19.177,152.182
C06102=1101.657,395.754,-93.842,179.881,19.171,152.181
C06103=1101.651,395.507,-93.804,179.878,19.165,152.180
C06104=1101.645,395.260,-93.766,179.876,19.159,152.179
C06105=1101.639,395.013,-93.729,179.873,19.154,152.178
C06106=1101.633,394.766,-93.691,179.870,19.148,152.177
C06107=1101.628,394.518,-93.653,179.868,19.142,152.176
C06108=1101.622,394.272,-93.615,179.866,19.136,152.175
C06109=1101.616,394.025,-93.578,179.863,19.130,152.174
C06110=1101.611,393.778,-93.540,179.861,19.125,152.173
C06111=1101.605,393.531,-93.503,179.858,19.118,152.172
C06112=1101.599,393.284,-93.465,179.856,19.112,152.171
C06113=1101.593,393.036,-93.426,179.853,19.107,152.171
C06114=1101.588,392.789,-93.389,179.851,19.101,152.169
C06115=1101.582,392.542,-93.352,179.848,19.095,152.168
C06116=1101.576,392.295,-93.315,179.846,19.090,152.168
C06117=1101.570,392.048,-93.277,179.843,19.084,152.167
C06118=1101.564,391.801,-93.239,179.840,19.078,152.166
C06119=1101.559,391.554,-93.202,179.838,19.073,152.165
C06120=1101.553,391.307,-93.164,179.835,19.067,152.164
C06121=1101.547,391.060,-93.127,179.833,19.062,152.163
C06122=1101.541,390.813,-93.089,179.830,19.056,152.162
C06123=1101.535,390.566,-93.053,179.828,19.050,152.161
C06124=1101.529,390.319,-93.015,179.825,19.044,152.160
C06125=1101.524,390.072,-92.978,179.822,19.039,152.159
C06126=1101.518,389.825,-92.941,179.819,19.034,152.159
C06127=1101.512,389.578,-92.903,179.817,19.028,152.158
C06128=1101.506,389.331,-92.866,179.814,19.023,152.157
C06129=1101.501,389.084,-92.829,179.812,19.017,152.156
C06130=1101.495,388.836,-92.792,179.809,19.012,152.155
C06131=1101.489,388.590,-92.754,179.807,19.006,152.154
C06132=1101.483,388.343,-92.717,179.804,19.001,152.153
C06133=1101.477,388.095,-92.680,179.801,18.995,152.152
C06134=1101.471,387.849,-92.643,179.799,18.990,152.152
C06135=1101.466,387.601,-92.606,179.796,18.985,152.151
C06136=1101.461,387.354,-92.569,179.793,18.979,152.150
C06137=1101.455,387.108,-92.531,179.791,18.974,152.149
C06138=1101.449,386.860,-92.494,179.788,18.969,152.148
C06139=1101.443,386.613,-92.458,179.785,18.963,152.147
C06140=1101.437,386.366,-92.421,179.783,18.958,152.147
C06141=1101.432,386.119,-92.384,179.780,18.953,152.146
C06142=1101.426,385.872,-92.346,179.778,18.947,152.145
C06143=1101.420,385.624,-92.309,179.775,18.942,152.144
C06144=1101.414,385.378,-92.273,179.772,18.937,152.143
C06145=1101.409,385.131,-92.236,179.770,18.931,152.142
C06146=1101.403,384.883,-92.199,179.767,18.926,152.142
C06147=1101.398,384.636,-92.162,179.765,18.921,152.141
C06148=1101.391,384.389,-92.125,179.762,18.916,152.140
C06149=1101.382,383.972,-92.063,179.757,18.907,152.139
C06150=1101.372,383.556,-92.001,179.753,18.898,152.138
C06151=1101.363,383.139,-91.938,179.748,18.889,152.136
C06152=1101.353,382.723,-91.876,179.744,18.881,152.135
C06153=1101.348,382.475,-91.839,179.741,18.876,152.134
C06154=1101.341,382.228,-91.803,179.738,18.871,152.133
C06155=1101.336,381.981,-91.766,179.735,18.866,152.133
C06156=1101.330,381.733,-91.730,179.733,18.861,152.132
C06157=1101.324,381.486,-91.693,179.730,18.856,152.131
C06158=1101.318,381.239,-91.657,179.727,18.851,152.131
C06159=1101.313,380.992,-91.620,179.724,18.846,152.130
C06160=1101.306,380.745,-91.584,179.721,18.841,152.129
C06161=1101.301,380.498,-91.547,179.719,18.836,152.129
C06162=1101.295,380.250,-91.510,179.716,18.831,152.128
C06163=1101.290,380.003,-91.474,179.714,18.827,152.127
C06164=1101.283,379.756,-91.438,179.711,18.822,152.126
C06165=1101.278,379.509,-91.401,179.708,18.817,152.126
C06166=1101.271,379.262,-91.364,179.705,18.812,152.125
C06167=1101.267,379.015,-91.328,179.702,18.807,152.124
C06168=1101.260,378.768,-91.292,179.700,18.802,152.124
C06169=1101.255,378.520,-91.255,179.697,18.797,152.123
C06170=1101.249,378.272,-91.219,179.694,18.793,152.122
C06171=1101.244,378.026,-91.182,179.691,18.788,152.122
C06172=1101.237,377.779,-91.146,179.688,18.783,152.121
C06173=1101.232,377.531,-91.110,179.686,18.779,152.120
C06174=1101.226,377.284,-91.074,179.683,18.774,152.120
C06175=1101.221,377.036,-91.037,179.681,18.769,152.119
C06176=1101.215,376.789,-91.001,179.678,18.764,152.119
C06177=1101.209,376.542,-90.965,179.675,18.759,152.118
C06178=1101.204,376.295,-90.928,179.672,18.755,152.117
C06179=1101.197,376.048,-90.892,179.669,18.750,152.117
C06180=1101.192,375.801,-90.857,179.666,18.745,152.116
C06181=1101.186,375.554,-90.820,179.664,18.741,152.115
C06182=1101.180,375.306,-90.784,179.661,18.736,152.115
C06183=1101.176,375.059,-90.748,179.658,18.731,152.114
C06184=1101.169,374.812,-90.711,179.655,18.727,152.113
C06185=1101.164,374.565,-90.676,179.652,18.722,152.113
C06186=1101.158,374.317,-90.639,179.649,18.717,152.112
C06187=1101.152,374.070,-90.603,179.647,18.713,152.112
C06188=1101.147,373.823,-90.568,179.644,18.709,152.111
C06189=1101.141,373.576,-90.531,179.641,18.704,152.111
C06190=1101.134,373.328,-90.496,179.638,18.699,152.110
C06191=1101.130,373.081,-90.460,179.635,18.695,152.109
C06192=1101.123,372.834,-90.423,179.633,18.691,152.109
C06193=1101.117,372.586,-90.388,179.630,18.686,152.108
C06194=1101.112,372.339,-90.352,179.627,18.681,152.108
C06195=1101.106,372.092,-90.316,179.624,18.677,152.107
C06196=1101.100,371.845,-90.280,179.621,18.673,152.107
C06197=1101.095,371.597,-90.244,179.618,18.669,152.106
C06198=1101.089,371.349,-90.208,179.615,18.664,152.106
C06199=1101.083,371.102,-90.173,179.613,18.659,152.105
C06200=1101.077,370.855,-90.137,179.609,18.655,152.105
C06201=1101.069,370.465,-90.081,179.605,18.648,152.104
C06202=1101.060,370.075,-90.024,179.600,18.641,152.103
C06203=1101.051,369.686,-89.968,179.596,18.634,152.102
C06204=1101.041,369.296,-89.912,179.591,18.628,152.101
C06205=1101.036,369.048,-89.876,179.589,18.624,152.101
C06206=1101.030,368.801,-89.841,179.586,18.619,152.100
C06207=1101.025,368.554,-89.805,179.583,18.615,152.100
C06208=1101.019,368.306,-89.769,179.580,18.611,152.099
C06209=1101.013,368.059,-89.734,179.577,18.606,152.099
C06210=1101.007,367.811,-89.698,179.574,18.602,152.098
C06211=1101.002,367.564,-89.663,179.571,18.598,152.098
C06212=1100.996,367.317,-89.627,179.569,18.594,152.097
C06213=1100.990,367.070,-89.592,179.566,18.589,152.097
C06214=1100.984,366.822,-89.556,179.562,18.585,152.096
C06215=1100.979,366.575,-89.521,179.560,18.581,152.096
C06216=1100.973,366.327,-89.485,179.557,18.577,152.095
C06217=1100.967,366.081,-89.450,179.554,18.573,152.095
C06218=1100.962,365.832,-89.415,179.551,18.568,152.094
C06219=1100.956,365.585,-89.379,179.548,18.565,152.094
C06220=1100.950,365.338,-89.344,179.545,18.561,152.093
C06221=1100.945,365.091,-89.308,179.542,18.556,152.093
C06222=1100.938,364.843,-89.273,179.540,18.552,152.092
C06223=1100.933,364.596,-89.238,179.536,18.548,152.092
C06224=1100.927,364.348,-89.203,179.533,18.544,152.092
C06225=1100.921,364.101,-89.167,179.531,18.540,152.091
C06226=1100.916,363.853,-89.133,179.527,18.536,152.091
C06227=1100.910,363.606,-89.097,179.524,18.532,152.090
C06228=1100.904,363.359,-89.062,179.522,18.528,152.090
C06229=1100.898,363.111,-89.027,179.519,18.524,152.090
C06230=1100.893,362.864,-88.992,179.515,18.520,152.089
C06231=1100.887,362.616,-88.956,179.513,18.516,152.089
C06232=1100.882,362.369,-88.922,179.509,18.512,152.088
C06233=1100.876,362.122,-88.887,179.507,18.509,152.088
C06234=1100.870,361.874,-88.851,179.504,18.504,152.088
C06235=1100.865,361.627,-88.816,179.501,18.500,152.087
C06236=1100.858,361.379,-88.781,179.498,18.496,152.087
C06237=1100.853,361.132,-88.747,179.495,18.493,152.086
C06238=1100.847,360.885,-88.711,179.491,18.488,152.086
C06239=1100.841,360.636,-88.676,179.489,18.485,152.086
C06240=1100.835,360.390,-88.641,179.486,18.480,152.085
C06241=1100.830,360.142,-88.607,179.483,18.477,152.085
C06242=1100.824,359.894,-88.571,179.480,18.473,152.084
C06243=1100.818,359.647,-88.537,179.477,18.469,152.084
C06244=1100.813,359.399,-88.502,179.474,18.466,152.084
C06245=1100.807,359.152,-88.467,179.471,18.461,152.083
C06246=1100.801,358.905,-88.433,179.468,18.458,152.083
C06247=1100.795,358.657,-88.397,179.465,18.454,152.083
C06248=1100.789,358.410,-88.363,179.462,18.451,152.082
C06249=1100.784,358.162,-88.328,179.459,18.446,152.082
C06250=1100.778,357.914,-88.292,179.455,18.443,152.082
C06251=1100.772,357.667,-88.258,179.453,18.439,152.081
C06252=1100.767,357.419,-88.224,179.450,18.435,152.081
C06253=1100.758,357.044,-88.171,179.445,18.429,152.080
C06254=1100.749,356.670,-88.119,179.440,18.424,152.080
C06255=1100.741,356.295,-88.066,179.436,18.419,152.079
C06256=1100.733,355.920,-88.014,179.432,18.413,152.079
C06257=1100.726,355.672,-87.979,179.428,18.409,152.079
C06258=1100.721,355.424,-87.944,179.426,18.406,152.078
C06259=1100.715,355.178,-87.910,179.422,18.402,152.078
C06260=1100.710,354.930,-87.875,179.419,18.398,152.078
C06261=1100.704,354.683,-87.841,179.416,18.394,152.077
C06262=1100.698,354.435,-87.806,179.413,18.391,152.077
C06263=1100.692,354.187,-87.772,179.410,18.387,152.077
C06264=1100.687,353.940,-87.738,179.407,18.384,152.077
C06265=1100.681,353.692,-87.703,179.404,18.380,152.076
C06266=1100.675,353.444,-87.669,179.401,18.376,152.076
C06267=1100.670,353.197,-87.634,179.398,18.373,152.076
C06268=1100.664,352.950,-87.600,179.395,18.369,152.075
C06269=1100.658,352.702,-87.566,179.392,18.366,152.075
C06270=1100.652,352.454,-87.531,179.389,18.362,152.075
C06271=1100.647,352.207,-87.497,179.386,18.359,152.074
C06272=1100.641,351.959,-87.463,179.382,18.355,152.074
C06273=1100.636,351.712,-87.428,179.380,18.352,152.074
C06274=1100.630,351.465,-87.394,179.376,18.348,152.074
C06275=1100.623,351.217,-87.360,179.374,18.345,152.073
C06276=1100.618,350.969,-87.325,179.370,18.341,152.073
C06277=1100.612,350.722,-87.291,179.367,18.338,152.073
C06278=1100.607,350.474,-87.258,179.364,18.335,152.073
C06279=1100.602,350.226,-87.223,179.361,18.331,152.072
C06280=1100.595,349.978,-87.189,179.358,18.328,152.072
C06281=1100.589,349.731,-87.155,179.355,18.324,152.072
C06282=1100.583,349.484,-87.121,179.352,18.321,152.072
C06283=1100.579,349.235,-87.087,179.348,18.317,152.072
C06284=1100.573,348.988,-87.053,179.346,18.314,152.071
C06285=1100.567,348.741,-87.019,179.342,18.310,152.071
C06286=1100.561,348.494,-86.985,179.340,18.307,152.071
C06287=1100.555,348.245,-86.951,179.336,18.304,152.071
C06288=1100.550,347.997,-86.916,179.333,18.300,152.070
C06289=1100.544,347.750,-86.882,179.331,18.297,152.070
C06290=1100.538,347.502,-86.849,179.327,18.294,152.070
C06291=1100.532,347.255,-86.815,179.324,18.291,152.070
C06292=1100.527,347.008,-86.781,179.321,18.287,152.069
C06293=1100.522,346.759,-86.747,179.318,18.284,152.069
C06294=1100.516,346.512,-86.713,179.314,18.280,152.069
C06295=1100.510,346.264,-86.679,179.311,18.277,152.069
C06296=1100.505,346.017,-86.645,179.309,18.274,152.069
C06297=1100.499,345.769,-86.612,179.305,18.271,152.069
C06298=1100.493,345.521,-86.578,179.302,18.267,152.068
C06299=1100.487,345.273,-86.544,179.299,18.264,152.068
C06300=1100.481,345.026,-86.510,179.296,18.261,152.068
C06301=1100.476,344.778,-86.477,179.293,18.258,152.068
C06302=1100.470,344.531,-86.443,179.289,18.254,152.068
C06303=1100.464,344.283,-86.409,179.287,18.251,152.067
C06304=1100.458,344.035,-86.375,179.283,18.247,152.067
C06305=1100.450,343.663,-86.324,179.279,18.243,152.067
C06306=1100.441,343.290,-86.274,179.274,18.238,152.067
C06307=1100.432,342.917,-86.224,179.269,18.234,152.066
C06308=1100.424,342.545,-86.173,179.264,18.229,152.066
C06309=1100.418,342.297,-86.139,179.261,18.226,152.066
C06310=1100.413,342.049,-86.105,179.258,18.222,152.066
C06311=1100.407,341.801,-86.072,179.255,18.220,152.066
C06312=1100.401,341.554,-86.039,179.252,18.217,152.066
C06313=1100.395,341.306,-86.006,179.248,18.213,152.065
C06314=1100.390,341.059,-85.972,179.245,18.210,152.065
C06315=1100.384,340.811,-85.939,179.243,18.207,152.065
C06316=1100.379,340.564,-85.906,179.239,18.204,152.065
C06317=1100.373,340.316,-85.872,179.236,18.201,152.065
C06318=1100.367,340.068,-85.838,179.233,18.198,152.065
C06319=1100.362,339.820,-85.805,179.230,18.194,152.065
C06320=1100.356,339.573,-85.771,179.227,18.192,152.064
C06321=1100.351,339.325,-85.738,179.224,18.189,152.064
C06322=1100.344,339.077,-85.705,179.220,18.185,152.064
C06323=1100.339,338.829,-85.672,179.217,18.183,152.064
C06324=1100.333,338.581,-85.639,179.214,18.180,152.064
C06325=1100.327,338.334,-85.605,179.210,18.176,152.064
C06326=1100.322,338.086,-85.571,179.207,18.173,152.064
C06327=1100.316,337.838,-85.539,179.204,18.171,152.064
C06328=1100.310,337.591,-85.505,179.202,18.168,152.064
C06329=1100.305,337.343,-85.472,179.198,18.164,152.063
C06330=1100.298,337.095,-85.439,179.195,18.162,152.063
C06331=1100.293,336.848,-85.406,179.192,18.159,152.063
C06332=1100.288,336.600,-85.373,179.188,18.155,152.063
C06333=1100.282,336.352,-85.340,179.185,18.153,152.063
C06334=1100.276,336.104,-85.307,179.182,18.150,152.063
C06335=1100.270,335.857,-85.273,179.179,18.147,152.063
C06336=1100.265,335.609,-85.240,179.175,18.144,152.063
C06337=1100.259,335.360,-85.208,179.173,18.141,152.063
C06338=1100.253,335.113,-85.175,179.170,18.138,152.063
C06339=1100.248,334.865,-85.142,179.167,18.136,152.062
C06340=1100.242,334.618,-85.109,179.163,18.133,152.062
C06341=1100.236,334.370,-85.076,179.160,18.130,152.062
C06342=1100.231,334.122,-85.042,179.157,18.127,152.062
C06343=1100.225,333.874,-85.010,179.153,18.123,152.062
C06344=1100.219,333.626,-84.977,179.150,18.121,152.062
C06345=1100.214,333.379,-84.945,179.147,18.118,152.062
C06346=1100.208,333.131,-84.911,179.144,18.115,152.062
C06347=1100.203,332.883,-84.878,179.140,18.112,152.062
C06348=1100.197,332.635,-84.846,179.137,18.110,152.062
C06349=1100.191,332.387,-84.813,179.134,18.107,152.062
C06350=1100.185,332.140,-84.780,179.131,18.104,152.062
C06351=1100.180,331.892,-84.747,179.128,18.102,152.062
C06352=1100.174,331.644,-84.715,179.124,18.098,152.062
C06353=1100.168,331.396,-84.681,179.121,18.096,152.062
C06354=1100.162,331.148,-84.649,179.118,18.093,152.062
C06355=1100.156,330.900,-84.617,179.115,18.091,152.062
C06356=1100.150,330.652,-84.583,179.112,18.088,152.062
C06357=1100.141,330.274,-84.534,179.107,18.084,152.062
C06358=1100.133,329.895,-84.484,179.102,18.080,152.061
C06359=1100.124,329.516,-84.434,179.096,18.075,152.061
C06360=1100.115,329.138,-84.385,179.092,18.071,152.061
C06361=1100.109,328.890,-84.352,179.089,18.069,152.061
C06362=1100.104,328.643,-84.320,179.086,18.066,152.061
C06363=1100.098,328.394,-84.288,179.082,18.063,152.061
C06364=1100.092,328.147,-84.254,179.079,18.061,152.061
C06365=1100.086,327.898,-84.222,179.076,18.058,152.061
C06366=1100.081,327.651,-84.190,179.072,18.056,152.061
C06367=1100.075,327.403,-84.158,179.069,18.053,152.061
C06368=1100.069,327.155,-84.124,179.066,18.050,152.061
C06369=1100.063,326.907,-84.092,179.062,18.047,152.061
C06370=1100.058,326.660,-84.061,179.059,18.045,152.061
C06371=1100.052,326.412,-84.027,179.056,18.042,152.061
C06372=1100.046,326.163,-83.995,179.053,18.040,152.061
C06373=1100.040,325.917,-83.963,179.050,18.037,152.061
C06374=1100.034,325.668,-83.931,179.047,18.035,152.061
C06375=1100.028,325.420,-83.899,179.043,18.032,152.061
C06376=1100.024,325.172,-83.867,179.040,18.029,152.061
C06377=1100.018,324.925,-83.834,179.037,18.027,152.061
C06378=1100.012,324.677,-83.802,179.033,18.024,152.061
C06379=1100.006,324.429,-83.770,179.030,18.022,152.061
C06380=1100.001,324.181,-83.737,179.027,18.019,152.061
C06381=1099.995,323.933,-83.705,179.024,18.017,152.061
C06382=1099.989,323.685,-83.673,179.021,18.014,152.061
C06383=1099.983,323.437,-83.641,179.017,18.011,152.061
C06384=1099.978,323.190,-83.610,179.014,18.009,152.062
C06385=1099.972,322.942,-83.576,179.011,18.006,152.061
C06386=1099.966,322.694,-83.544,179.008,18.004,152.061
C06387=1099.961,322.446,-83.513,179.004,18.001,152.061
C06388=1099.955,322.198,-83.481,179.001,17.999,152.062
C06389=1099.950,321.950,-83.449,178.998,17.997,152.062
C06390=1099.944,321.702,-83.417,178.995,17.994,152.062
C06391=1099.938,321.455,-83.385,178.991,17.991,152.062
C06392=1099.933,321.206,-83.353,178.988,17.989,152.062
C06393=1099.928,320.959,-83.321,178.985,17.986,152.062
C06394=1099.922,320.710,-83.289,178.981,17.984,152.062
C06395=1099.916,320.462,-83.257,178.978,17.981,152.062
C06396=1099.910,320.215,-83.224,178.975,17.979,152.062
C06397=1099.904,319.967,-83.192,178.972,17.977,152.062
C06398=1099.899,319.719,-83.162,178.969,17.974,152.062
C06399=1099.893,319.471,-83.129,178.966,17.972,152.062
C06400=1099.887,319.223,-83.098,178.962,17.969,152.062
C06401=1099.881,318.975,-83.066,178.959,17.967,152.062
C06402=1099.877,318.727,-83.034,178.955,17.964,152.062
C06403=1099.871,318.480,-83.002,178.952,17.962,152.062
C06404=1099.865,318.231,-82.970,178.949,17.959,152.062
C06405=1099.860,317.984,-82.938,178.946,17.957,152.062
C06406=1099.854,317.736,-82.906,178.942,17.954,152.062
C06407=1099.849,317.488,-82.874,178.939,17.952,152.062
C06408=1099.843,317.240,-82.842,178.936,17.950,152.062
C06409=1099.834,316.854,-82.795,178.931,17.946,152.062
C06410=1099.826,316.469,-82.745,178.926,17.942,152.062
C06411=1099.817,316.083,-82.695,178.921,17.938,152.063
C06412=1099.808,315.697,-82.646,178.916,17.935,152.063
C06413=1099.803,315.449,-82.614,178.913,17.932,152.063
C06414=1099.797,315.201,-82.584,178.909,17.930,152.063
C06415=1099.791,314.953,-82.552,178.906,17.928,152.063
C06416=1099.786,314.706,-82.520,178.903,17.926,152.063
C06417=1099.780,314.458,-82.488,178.900,17.924,152.063
C06418=1099.774,314.210,-82.458,178.896,17.921,152.063
C06419=1099.768,313.961,-82.426,178.892,17.918,152.063
C06420=1099.763,313.714,-82.394,178.889,17.916,152.063
C06421=1099.756,313.465,-82.363,178.886,17.914,152.064
C06422=1099.751,313.218,-82.332,178.882,17.912,152.064
C06423=1099.745,312.969,-82.300,178.879,17.910,152.064
C06424=1099.739,312.722,-82.269,178.876,17.908,152.064
C06425=1099.734,312.474,-82.238,178.872,17.905,152.064
C06426=1099.728,312.226,-82.206,178.869,17.903,152.064
C06427=1099.722,311.978,-82.175,178.866,17.901,152.064
C06428=1099.716,311.730,-82.144,178.863,17.898,152.064
C06429=1099.710,311.482,-82.113,178.859,17.896,152.065
C06430=1099.705,311.234,-82.082,178.856,17.894,152.065
C06431=1099.699,310.986,-82.050,178.852,17.892,152.065
C06432=1099.693,310.738,-82.019,178.849,17.890,152.065
C06433=1099.688,310.491,-81.988,178.846,17.888,152.065
C06434=1099.681,310.242,-81.957,178.843,17.885,152.065
C06435=1099.676,309.995,-81.925,178.839,17.883,152.065
C06436=1099.671,309.746,-81.894,178.836,17.881,152.065
C06437=1099.664,309.499,-81.863,178.832,17.879,152.066
C06438=1099.659,309.250,-81.832,178.829,17.877,152.066
C06439=1099.653,309.003,-81.802,178.826,17.875,152.066
C06440=1099.647,308.754,-81.770,178.823,17.872,152.066
C06441=1099.642,308.507,-81.739,178.819,17.870,152.066
C06442=1099.636,308.258,-81.708,178.816,17.868,152.066
C06443=1099.630,308.011,-81.677,178.813,17.866,152.066
C06444=1099.625,307.762,-81.646,178.809,17.864,152.066
C06445=1099.619,307.515,-81.616,178.806,17.862,152.067
C06446=1099.613,307.267,-81.584,178.802,17.860,152.067
C06447=1099.608,307.018,-81.553,178.799,17.857,152.067
C06448=1099.602,306.770,-81.522,178.797,17.856,152.067
C06449=1099.596,306.523,-81.491,178.793,17.854,152.067
C06450=1099.591,306.275,-81.460,178.790,17.852,152.067
C06451=1099.585,306.027,-81.430,178.786,17.850,152.067
C06452=1099.579,305.778,-81.399,178.783,17.847,152.068
C06453=1099.573,305.531,-81.368,178.780,17.845,152.068
C06454=1099.568,305.283,-81.337,178.777,17.843,152.068
C06455=1099.562,305.035,-81.306,178.773,17.841,152.068
C06456=1099.557,304.787,-81.275,178.770,17.839,152.068
C06457=1099.551,304.539,-81.245,178.766,17.837,152.068
C06458=1099.546,304.290,-81.214,178.763,17.835,152.068
C06459=1099.540,304.043,-81.183,178.760,17.833,152.069
C06460=1099.534,303.795,-81.153,178.756,17.830,152.069
C06461=1099.525,303.412,-81.105,178.751,17.827,152.069
C06462=1099.517,303.029,-81.057,178.746,17.824,152.069
C06463=1099.508,302.645,-81.010,178.741,17.821,152.069
C06464=1099.499,302.263,-80.963,178.735,17.817,152.070
C06465=1099.494,302.014,-80.932,178.732,17.815,152.070
C06466=1099.488,301.767,-80.902,178.729,17.814,152.070
C06467=1099.483,301.519,-80.871,178.726,17.811,152.070
C06468=1099.477,301.271,-80.841,178.723,17.809,152.070
C06469=1099.472,301.023,-80.810,178.719,17.807,152.071
C06470=1099.467,300.775,-80.779,178.716,17.805,152.071
C06471=1099.461,300.526,-80.750,178.712,17.803,152.071
C06472=1099.455,300.278,-80.719,178.709,17.801,152.071
C06473=1099.450,300.030,-80.688,178.705,17.799,152.071
C06474=1099.444,299.782,-80.658,178.702,17.797,152.071
C06475=1099.438,299.534,-80.627,178.699,17.795,152.072
C06476=1099.433,299.286,-80.596,178.695,17.793,152.072
C06477=1099.427,299.038,-80.566,178.692,17.791,152.072
C06478=1099.422,298.790,-80.536,178.689,17.789,152.072
C06479=1099.416,298.541,-80.505,178.685,17.787,152.072
C06480=1099.411,298.294,-80.475,178.683,17.785,152.072
C06481=1099.405,298.046,-80.445,178.679,17.783,152.073
C06482=1099.399,297.797,-80.415,178.676,17.781,152.073
C06483=1099.393,297.550,-80.385,178.672,17.779,152.073
C06484=1099.388,297.302,-80.354,178.669,17.777,152.073
C06485=1099.382,297.054,-80.324,178.666,17.775,152.073
C06486=1099.377,296.805,-80.294,178.662,17.773,152.074
C06487=1099.371,296.557,-80.263,178.659,17.771,152.074
C06488=1099.365,296.310,-80.233,178.655,17.769,152.074
C06489=1099.360,296.061,-80.203,178.652,17.768,152.074
C06490=1099.354,295.813,-80.173,178.649,17.766,152.074
C06491=1099.348,295.565,-80.143,178.646,17.764,152.075
C06492=1099.343,295.317,-80.113,178.642,17.762,152.075
C06493=1099.337,295.069,-80.083,178.639,17.760,152.075
C06494=1099.331,294.821,-80.053,178.635,17.758,152.075
C06495=1099.326,294.573,-80.023,178.632,17.756,152.075
C06496=1099.320,294.324,-79.993,178.628,17.754,152.076
C06497=1099.314,294.077,-79.963,178.626,17.753,152.076
C06498=1099.309,293.828,-79.933,178.622,17.751,152.076
C06499=1099.303,293.580,-79.903,178.619,17.749,152.076
C06500=1099.297,293.333,-79.872,178.615,17.747,152.076
C06501=1099.292,293.084,-79.843,178.612,17.745,152.077
C06502=1099.286,292.836,-79.813,178.608,17.743,152.077
C06503=1099.280,292.588,-79.783,178.605,17.741,152.077
C06504=1099.275,292.339,-79.753,178.602,17.740,152.077
C06505=1099.269,292.092,-79.723,178.598,17.738,152.078
C06506=1099.263,291.843,-79.693,178.595,17.736,152.078
C06507=1099.258,291.596,-79.663,178.591,17.734,152.078
C06508=1099.252,291.348,-79.634,178.588,17.732,152.078
C06509=1099.247,291.099,-79.605,178.585,17.730,152.079
C06510=1099.241,290.852,-79.574,178.582,17.729,152.079
C06511=1099.235,290.603,-79.545,178.578,17.727,152.079
C06512=1099.230,290.355,-79.515,178.575,17.725,152.079
C06513=1099.221,289.986,-79.470,178.570,17.722,152.080
C06514=1099.213,289.616,-79.427,178.564,17.720,152.080
C06515=1099.204,289.247,-79.382,178.560,17.718,152.080
C06516=1099.196,288.878,-79.339,178.555,17.714,152.081
C06517=1099.190,288.630,-79.308,178.551,17.713,152.081
C06518=1099.184,288.382,-79.279,178.547,17.711,152.081
C06519=1099.179,288.133,-79.249,178.545,17.710,152.081
C06520=1099.173,287.885,-79.220,178.541,17.708,152.082
C06521=1099.167,287.637,-79.190,178.538,17.706,152.082
C06522=1099.162,287.388,-79.161,178.534,17.704,152.082
C06523=1099.156,287.141,-79.131,178.531,17.702,152.082
C06524=1099.150,286.893,-79.102,178.528,17.701,152.083
C06525=1099.145,286.645,-79.072,178.524,17.699,152.083
C06526=1099.139,286.396,-79.042,178.521,17.697,152.083
C06527=1099.133,286.148,-79.013,178.517,17.695,152.083
C06528=1099.127,285.900,-78.984,178.514,17.694,152.084
C06529=1099.122,285.652,-78.955,178.511,17.693,152.084
C06530=1099.116,285.404,-78.925,178.507,17.691,152.084
C06531=1099.111,285.155,-78.896,178.504,17.689,152.084
C06532=1099.105,284.907,-78.866,178.501,17.687,152.085
C06533=1099.099,284.659,-78.837,178.497,17.685,152.085
C06534=1099.094,284.411,-78.808,178.494,17.684,152.085
C06535=1099.088,284.163,-78.778,178.491,17.682,152.085
C06536=1099.082,283.914,-78.749,178.487,17.680,152.086
C06537=1099.077,283.666,-78.720,178.483,17.679,152.086
C06538=1099.071,283.418,-78.690,178.481,17.677,152.086
C06539=1099.066,283.170,-78.661,178.477,17.675,152.086
C06540=1099.060,282.922,-78.632,178.474,17.674,152.087
C06541=1099.054,282.674,-78.603,178.470,17.672,152.087
C06542=1099.049,282.426,-78.573,178.467,17.670,152.087
C06543=1099.043,282.177,-78.544,178.464,17.669,152.088
C06544=1099.037,281.929,-78.515,178.460,17.667,152.088
C06545=1099.032,281.680,-78.486,178.457,17.665,152.088
C06546=1099.026,281.433,-78.457,178.453,17.663,152.088
C06547=1099.021,281.184,-78.427,178.450,17.662,152.089
C06548=1099.015,280.936,-78.398,178.447,17.660,152.089
C06549=1099.009,280.687,-78.369,178.443,17.659,152.089
C06550=1099.004,280.440,-78.341,178.440,17.657,152.089
C06551=1098.998,280.191,-78.311,178.437,17.656,152.090
C06552=1098.992,279.943,-78.282,178.433,17.654,152.090
C06553=1098.987,279.695,-78.254,178.430,17.652,152.090
C06554=1098.981,279.447,-78.225,178.426,17.650,152.091
C06555=1098.976,279.198,-78.195,178.423,17.649,152.091
C06556=1098.969,278.950,-78.166,178.420,17.648,152.091
C06557=1098.964,278.702,-78.138,178.416,17.646,152.091
C06558=1098.958,278.454,-78.108,178.412,17.644,152.092
C06559=1098.952,278.205,-78.079,178.410,17.643,152.092
C06560=1098.948,277.957,-78.051,178.406,17.641,152.092
C06561=1098.941,277.709,-78.022,178.403,17.639,152.093
C06562=1098.935,277.460,-77.993,178.399,17.638,152.093
C06563=1098.930,277.212,-77.964,178.396,17.636,152.093
C06564=1098.924,276.964,-77.935,178.393,17.635,152.093
C06565=1098.916,276.604,-77.894,178.387,17.632,152.094
C06566=1098.908,276.244,-77.851,178.383,17.630,152.094
C06567=1098.900,275.884,-77.810,178.378,17.628,152.095
C06568=1098.892,275.525,-77.768,178.373,17.625,152.095
C06569=1098.886,275.276,-77.740,178.370,17.624,152.096
C06570=1098.881,275.029,-77.711,178.366,17.623,152.096
C06571=1098.875,274.780,-77.683,178.362,17.621,152.096
C06572=1098.869,274.531,-77.654,178.359,17.619,152.096
C06573=1098.864,274.283,-77.625,178.356,17.618,152.097
C06574=1098.858,274.035,-77.597,178.353,17.616,152.097
C06575=1098.853,273.787,-77.568,178.349,17.615,152.097
C06576=1098.847,273.538,-77.539,178.346,17.613,152.098
C06577=1098.841,273.289,-77.511,178.342,17.612,152.098
C06578=1098.835,273.042,-77.482,178.339,17.610,152.098
C06579=1098.829,272.793,-77.454,178.335,17.608,152.099
C06580=1098.824,272.546,-77.425,178.332,17.608,152.099
C06581=1098.819,272.297,-77.396,178.329,17.606,152.099
C06582=1098.813,272.049,-77.368,178.325,17.604,152.100
C06583=1098.807,271.800,-77.340,178.322,17.603,152.100
C06584=1098.801,271.552,-77.311,178.319,17.601,152.100
C06585=1098.796,271.304,-77.283,178.315,17.600,152.101
C06586=1098.790,271.055,-77.255,178.312,17.598,152.101
C06587=1098.785,270.807,-77.226,178.309,17.597,152.101
C06588=1098.779,270.559,-77.197,178.305,17.595,152.101
C06589=1098.774,270.310,-77.169,178.302,17.594,152.102
C06590=1098.768,270.062,-77.141,178.298,17.593,152.102
C06591=1098.762,269.814,-77.113,178.295,17.591,152.102
C06592=1098.756,269.565,-77.085,178.291,17.589,152.103
C06593=1098.751,269.317,-77.056,178.288,17.588,152.103
C06594=1098.745,269.069,-77.028,178.285,17.586,152.103
C06595=1098.739,268.821,-77.000,178.281,17.585,152.104
C06596=1098.733,268.572,-76.971,178.278,17.584,152.104
C06597=1098.728,268.324,-76.943,178.274,17.582,152.104
C06598=1098.722,268.075,-76.915,178.271,17.580,152.105
C06599=1098.717,267.827,-76.887,178.268,17.580,152.105
C06600=1098.711,267.578,-76.859,178.264,17.578,152.105
C06601=1098.705,267.330,-76.831,178.261,17.576,152.106
C06602=1098.700,267.082,-76.802,178.258,17.575,152.106
C06603=1098.694,266.833,-76.775,178.254,17.574,152.106
C06604=1098.688,266.585,-76.746,178.251,17.572,152.107
C06605=1098.683,266.337,-76.718,178.248,17.571,152.107
C06606=1098.678,266.089,-76.690,178.244,17.569,152.107
C06607=1098.672,265.840,-76.662,178.240,17.567,152.108
C06608=1098.666,265.592,-76.634,178.237,17.566,152.108
C06609=1098.660,265.343,-76.606,178.234,17.565,152.108
C06610=1098.655,265.095,-76.578,178.230,17.564,152.109
C06611=1098.649,264.846,-76.549,178.227,17.562,152.109
C06612=1098.644,264.598,-76.521,178.223,17.561,152.109
C06613=1098.638,264.350,-76.494,178.221,17.560,152.110
C06614=1098.632,264.102,-76.466,178.217,17.558,152.110
C06615=1098.626,263.854,-76.438,178.213,17.556,152.110
C06616=1098.621,263.604,-76.410,178.210,17.555,152.111
C06617=1098.612,263.248,-76.370,178.205,17.553,152.111
C06618=1098.604,262.891,-76.330,178.200,17.552,152.112
C06619=1098.596,262.534,-76.290,178.195,17.549,152.112
C06620=1098.587,262.177,-76.250,178.191,17.548,152.113
C06621=1098.582,261.928,-76.223,178.187,17.546,152.113
C06622=1098.576,261.679,-76.195,178.184,17.545,152.114
C06623=1098.571,261.431,-76.167,178.180,17.544,152.114
C06624=1098.564,261.183,-76.139,178.177,17.542,152.114
C06625=1098.559,260.934,-76.112,178.174,17.541,152.115
C06626=1098.554,260.686,-76.084,178.170,17.540,152.115
C06627=1098.547,260.438,-76.056,178.166,17.538,152.115
C06628=1098.542,260.189,-76.029,178.163,17.537,152.116
C06629=1098.536,259.940,-76.000,178.160,17.536,152.116
C06630=1098.530,259.692,-75.973,178.157,17.535,152.116
C06631=1098.525,259.444,-75.946,178.153,17.533,152.117
C06632=1098.518,259.195,-75.918,178.149,17.532,152.117
C06633=1098.513,258.947,-75.890,178.146,17.531,152.117
C06634=1098.508,258.699,-75.863,178.143,17.529,152.118
C06635=1098.501,258.450,-75.835,178.140,17.528,152.118
C06636=1098.496,258.201,-75.808,178.136,17.527,152.119
C06637=1098.491,257.953,-75.780,178.132,17.525,152.119
C06638=1098.485,257.705,-75.753,178.129,17.524,152.119
C06639=1098.479,257.456,-75.725,178.126,17.523,152.120
C06640=1098.473,257.208,-75.698,178.123,17.522,152.120
C06641=1098.468,256.960,-75.670,178.119,17.520,152.120
C06642=1098.462,256.711,-75.643,178.115,17.518,152.121
C06643=1098.456,256.463,-75.615,178.112,17.518,152.121
C06644=1098.451,256.214,-75.588,178.109,17.516,152.121
C06645=1098.445,255.966,-75.561,178.106,17.515,152.122
C06646=1098.439,255.717,-75.533,178.102,17.514,152.122
C06647=1098.434,255.469,-75.507,178.098,17.512,152.123
C06648=1098.428,255.221,-75.479,178.095,17.511,152.123
C06649=1098.423,254.972,-75.452,178.092,17.510,152.123
C06650=1098.417,254.723,-75.424,178.089,17.509,152.124
C06651=1098.411,254.475,-75.397,178.085,17.507,152.124
C06652=1098.406,254.226,-75.370,178.082,17.506,152.124
C06653=1098.400,253.979,-75.342,178.078,17.505,152.125
C06654=1098.395,253.730,-75.315,178.075,17.503,152.125
C06655=1098.389,253.481,-75.287,178.072,17.502,152.126
C06656=1098.383,253.233,-75.260,178.068,17.501,152.126
C06657=1098.378,252.984,-75.233,178.065,17.500,152.126
C06658=1098.372,252.736,-75.206,178.062,17.498,152.127
C06659=1098.366,252.488,-75.180,178.058,17.496,152.127
C06660=1098.361,252.239,-75.152,178.055,17.496,152.127
C06661=1098.355,251.990,-75.125,178.051,17.494,152.128
C06662=1098.350,251.742,-75.097,178.048,17.493,152.128
C06663=1098.344,251.493,-75.071,178.044,17.492,152.128
C06664=1098.339,251.245,-75.043,178.041,17.491,152.129
C06665=1098.333,250.996,-75.017,178.038,17.489,152.129
C06666=1098.328,250.748,-74.989,178.035,17.488,152.130
C06667=1098.322,250.500,-74.962,178.031,17.487,152.130
C06668=1098.317,250.251,-74.935,178.027,17.485,152.130
C06669=1098.309,249.890,-74.896,178.023,17.483,152.131
C06670=1098.301,249.531,-74.857,178.018,17.482,152.131
C06671=1098.292,249.170,-74.818,178.013,17.480,152.132
C06672=1098.285,248.811,-74.779,178.008,17.478,152.132
C06673=1098.279,248.562,-74.752,178.005,17.477,152.133
C06674=1098.273,248.314,-74.725,178.002,17.476,152.133
C06675=1098.268,248.065,-74.698,177.998,17.474,152.134
C06676=1098.262,247.817,-74.671,177.995,17.473,152.134
C06677=1098.256,247.569,-74.645,177.991,17.472,152.134
C06678=1098.251,247.320,-74.617,177.988,17.471,152.135
C06679=1098.246,247.072,-74.591,177.985,17.470,152.135
C06680=1098.239,246.823,-74.564,177.981,17.468,152.135
C06681=1098.233,246.574,-74.537,177.978,17.467,152.136
C06682=1098.228,246.326,-74.510,177.974,17.466,152.136
C06683=1098.223,246.077,-74.483,177.971,17.465,152.137
C06684=1098.217,245.828,-74.457,177.967,17.463,152.137
C06685=1098.211,245.580,-74.431,177.964,17.462,152.137
C06686=1098.206,245.331,-74.403,177.961,17.461,152.138
C06687=1098.201,245.083,-74.377,177.958,17.460,152.138
C06688=1098.195,244.834,-74.350,177.954,17.459,152.139
C06689=1098.189,244.586,-74.323,177.951,17.458,152.139
C06690=1098.183,244.338,-74.297,177.947,17.456,152.139
C06691=1098.178,244.089,-74.271,177.944,17.455,152.140
C06692=1098.173,243.840,-74.244,177.941,17.453,152.140
C06693=1098.167,243.592,-74.217,177.938,17.453,152.140
C06694=1098.161,243.343,-74.190,177.934,17.451,152.141
C06695=1098.156,243.094,-74.164,177.931,17.451,152.141
C06696=1098.150,242.846,-74.138,177.927,17.449,152.142
C06697=1098.144,242.598,-74.111,177.924,17.448,152.142
C06698=1098.138,242.349,-74.084,177.921,17.447,152.142
C06699=1098.133,242.100,-74.059,177.918,17.446,152.143
C06700=1098.127,241.852,-74.032,177.914,17.444,152.143
C06701=1098.121,241.604,-74.005,177.911,17.444,152.144
C06702=1098.116,241.355,-73.979,177.907,17.442,152.144
C06703=1098.110,241.106,-73.953,177.904,17.441,152.144
C06704=1098.104,240.858,-73.926,177.900,17.440,152.145
C06705=1098.099,240.609,-73.900,177.897,17.439,152.145
C06706=1098.093,240.361,-73.873,177.894,17.437,152.146
C06707=1098.087,240.112,-73.847,177.891,17.437,152.146
C06708=1098.082,239.863,-73.821,177.887,17.436,152.146
C06709=1098.076,239.615,-73.794,177.884,17.435,152.147
C06710=1098.071,239.366,-73.768,177.880,17.433,152.147
C06711=1098.066,239.118,-73.742,177.877,17.432,152.148
C06712=1098.060,238.869,-73.716,177.873,17.431,152.148
C06713=1098.054,238.621,-73.689,177.870,17.430,152.148
C06714=1098.049,238.372,-73.663,177.867,17.428,152.149
C06715=1098.043,238.124,-73.637,177.864,17.428,152.149
C06716=1098.038,237.875,-73.611,177.860,17.426,152.150
C06717=1098.031,237.627,-73.585,177.857,17.425,152.150
C06718=1098.026,237.378,-73.559,177.853,17.424,152.151
C06719=1098.020,237.129,-73.532,177.850,17.423,152.151
C06720=1098.014,236.880,-73.506,177.846,17.422,152.151
C06721=1098.006,236.513,-73.468,177.841,17.420,152.152
C06722=1097.998,236.147,-73.429,177.837,17.419,152.152
C06723=1097.990,235.780,-73.391,177.832,17.417,152.153
C06724=1097.982,235.413,-73.352,177.827,17.415,152.154
C06725=1097.976,235.165,-73.327,177.824,17.415,152.154
C06726=1097.970,234.916,-73.301,177.820,17.413,152.154
C06727=1097.964,234.667,-73.274,177.817,17.412,152.155
C06728=1097.959,234.418,-73.248,177.813,17.411,152.155
C06729=1097.954,234.169,-73.222,177.810,17.410,152.156
C06730=1097.949,233.921,-73.197,177.806,17.409,152.156
C06731=1097.942,233.673,-73.171,177.803,17.408,152.157
C06732=1097.937,233.424,-73.145,177.800,17.407,152.157
C06733=1097.931,233.175,-73.119,177.797,17.406,152.157
C06734=1097.926,232.926,-73.093,177.794,17.405,152.158
C06735=1097.920,232.679,-73.067,177.790,17.403,152.158
C06736=1097.914,232.430,-73.041,177.787,17.402,152.158
C06737=1097.909,232.181,-73.015,177.783,17.401,152.159
C06738=1097.903,231.932,-72.990,177.780,17.401,152.159
C06739=1097.897,231.683,-72.964,177.776,17.399,152.160
C06740=1097.892,231.435,-72.938,177.773,17.398,152.160
C06741=1097.887,231.187,-72.912,177.770,17.397,152.161
C06742=1097.880,230.938,-72.886,177.767,17.396,152.161
C06743=1097.875,230.689,-72.860,177.764,17.395,152.161
C06744=1097.870,230.441,-72.835,177.760,17.394,152.162
C06745=1097.864,230.192,-72.810,177.757,17.393,152.162
C06746=1097.858,229.943,-72.784,177.753,17.392,152.163
C06747=1097.852,229.694,-72.758,177.750,17.391,152.163
C06748=1097.847,229.446,-72.733,177.747,17.390,152.163
C06749=1097.841,229.197,-72.707,177.743,17.388,152.164
C06750=1097.836,228.948,-72.681,177.740,17.388,152.164
C06751=1097.829,228.700,-72.656,177.736,17.387,152.165
C06752=1097.825,228.451,-72.631,177.733,17.386,152.165
C06753=1097.818,228.203,-72.605,177.730,17.384,152.166
C06754=1097.813,227.954,-72.579,177.727,17.383,152.166
C06755=1097.807,227.705,-72.553,177.723,17.383,152.167
C06756=1097.802,227.457,-72.528,177.720,17.382,152.167
C06757=1097.796,227.208,-72.502,177.717,17.381,152.167
C06758=1097.790,226.959,-72.477,177.713,17.379,152.168
C06759=1097.785,226.711,-72.452,177.710,17.378,152.168
C06760=1097.779,226.462,-72.426,177.707,17.377,152.169
C06761=1097.773,226.214,-72.401,177.703,17.376,152.169
C06762=1097.768,225.965,-72.375,177.700,17.376,152.169
C06763=1097.762,225.717,-72.350,177.696,17.374,152.170
C06764=1097.757,225.467,-72.325,177.693,17.373,152.170
C06765=1097.751,225.219,-72.300,177.690,17.372,152.171
C06766=1097.746,224.970,-72.274,177.686,17.371,152.171
C06767=1097.739,224.721,-72.248,177.683,17.371,152.172
C06768=1097.735,224.473,-72.223,177.680,17.369,152.172
C06769=1097.728,224.224,-72.198,177.677,17.368,152.172
C06770=1097.723,223.975,-72.172,177.674,17.367,152.173
C06771=1097.718,223.727,-72.147,177.670,17.366,152.173
C06772=1097.711,223.478,-72.122,177.667,17.365,152.174
C06773=1097.703,223.103,-72.084,177.662,17.364,152.174
C06774=1097.695,222.727,-72.046,177.657,17.362,152.175
C06775=1097.686,222.353,-72.008,177.652,17.361,152.175
C06776=1097.678,221.976,-71.970,177.647,17.360,152.176
C06777=1097.673,221.727,-71.945,177.643,17.358,152.177
C06778=1097.667,221.479,-71.919,177.640,17.357,152.177
C06779=1097.661,221.230,-71.894,177.637,17.356,152.177
C06780=1097.655,220.982,-71.870,177.633,17.355,152.178
C06781=1097.650,220.733,-71.844,177.630,17.355,152.178
C06782=1097.644,220.485,-71.819,177.627,17.353,152.179
C06783=1097.638,220.235,-71.794,177.624,17.352,152.179
C06784=1097.632,219.987,-71.769,177.620,17.352,152.180
C06785=1097.627,219.738,-71.745,177.617,17.350,152.180
C06786=1097.621,219.489,-71.719,177.614,17.349,152.181
C06787=1097.616,219.240,-71.695,177.611,17.349,152.181
C06788=1097.610,218.992,-71.669,177.607,17.348,152.181
C06789=1097.605,218.743,-71.645,177.604,17.347,152.182
C06790=1097.598,218.495,-71.620,177.601,17.346,152.182
C06791=1097.594,218.246,-71.595,177.597,17.344,152.183
C06792=1097.588,217.997,-71.569,177.594,17.344,152.183
C06793=1097.582,217.748,-71.545,177.590,17.343,152.184
C06794=1097.576,217.500,-71.520,177.587,17.342,152.184
C06795=1097.571,217.251,-71.496,177.584,17.341,152.184
C06796=1097.565,217.002,-71.470,177.580,17.340,152.185
C06797=1097.560,216.754,-71.445,177.577,17.339,152.185
C06798=1097.554,216.505,-71.420,177.574,17.338,152.186
C06799=1097.549,216.256,-71.396,177.570,17.337,152.186
C06800=1097.543,216.007,-71.371,177.567,17.336,152.187
C06801=1097.537,215.759,-71.346,177.564,17.335,152.187
C06802=1097.531,215.510,-71.322,177.560,17.334,152.187
C06803=1097.526,215.261,-71.297,177.557,17.333,152.188
C06804=1097.520,215.012,-71.271,177.555,17.332,152.188
C06805=1097.515,214.764,-71.247,177.550,17.331,152.189
C06806=1097.510,214.515,-71.223,177.548,17.330,152.189
C06807=1097.504,214.266,-71.198,177.545,17.330,152.190
C06808=1097.498,214.018,-71.173,177.541,17.328,152.190
C06809=1097.492,213.768,-71.149,177.538,17.327,152.190
C06810=1097.487,213.521,-71.124,177.535,17.327,152.191
C06811=1097.481,213.271,-71.099,177.531,17.325,152.191
C06812=1097.476,213.023,-71.075,177.528,17.325,152.192
C06813=1097.470,212.774,-71.051,177.525,17.324,152.192
C06814=1097.464,212.525,-71.026,177.522,17.323,152.193
C06815=1097.459,212.277,-71.001,177.518,17.322,152.193
C06816=1097.453,212.028,-70.976,177.515,17.321,152.194
C06817=1097.448,211.779,-70.952,177.512,17.320,152.194
C06818=1097.442,211.530,-70.928,177.508,17.319,152.194
C06819=1097.436,211.281,-70.903,177.505,17.318,152.195
C06820=1097.431,211.032,-70.879,177.502,17.317,152.195
C06821=1097.425,210.784,-70.854,177.498,17.316,152.196
C06822=1097.420,210.535,-70.829,177.495,17.316,152.196
C06823=1097.414,210.287,-70.805,177.492,17.315,152.197
C06824=1097.408,210.037,-70.780,177.488,17.313,152.197
C06825=1097.400,209.666,-70.745,177.484,17.313,152.198
C06826=1097.392,209.295,-70.708,177.479,17.311,152.198
C06827=1097.383,208.923,-70.672,177.474,17.310,152.199
C06828=1097.375,208.551,-70.635,177.469,17.309,152.200
C06829=1097.351,207.540,-70.538,177.422,17.291,152.205
C06830=1097.346,207.291,-70.513,177.419,17.291,152.206
C06831=1097.341,207.042,-70.489,177.415,17.291,152.206
C06832=1097.335,206.793,-70.466,177.412,17.290,152.207
C06833=1097.329,206.544,-70.441,177.408,17.290,152.208
C06834=1097.324,206.296,-70.417,177.405,17.290,152.208
C06835=1097.318,206.047,-70.394,177.401,17.291,152.209
C06836=1097.313,205.799,-70.369,177.398,17.290,152.210
C06837=1097.307,205.549,-70.345,177.394,17.290,152.210
C06838=1097.301,205.301,-70.322,177.391,17.290,152.211
C06839=1097.296,205.052,-70.298,177.388,17.290,152.212
C06840=1097.290,204.803,-70.273,177.384,17.290,152.212
C06841=1097.285,204.554,-70.250,177.381,17.290,152.213
C06842=1097.279,204.305,-70.226,177.377,17.290,152.214
C06843=1097.273,204.057,-70.202,177.374,17.290,152.214
C06844=1097.268,203.808,-70.178,177.370,17.290,152.215
C06845=1097.262,203.559,-70.154,177.367,17.290,152.216
C06846=1097.256,203.311,-70.131,177.364,17.289,152.216
C06847=1097.251,203.061,-70.107,177.360,17.290,152.217
C06848=1097.245,202.813,-70.083,177.357,17.290,152.218
C06849=1097.240,202.563,-70.059,177.353,17.289,152.218
C06850=1097.234,202.315,-70.036,177.350,17.289,152.219
C06851=1097.228,202.067,-70.012,177.346,17.289,152.220
C06852=1097.222,201.817,-69.988,177.343,17.289,152.220
C06853=1097.217,201.568,-69.964,177.339,17.289,152.221
C06854=1097.211,201.320,-69.941,177.336,17.289,152.222
C06855=1097.205,201.071,-69.917,177.332,17.289,152.222
C06856=1097.200,200.823,-69.893,177.329,17.289,152.223
C06857=1097.193,200.573,-69.870,177.326,17.289,152.223
C06858=1097.188,200.324,-69.846,177.322,17.289,152.224
C06859=1097.182,200.076,-69.823,177.319,17.289,152.225
C06860=1097.176,199.827,-69.799,177.315,17.289,152.225
C06861=1097.171,199.578,-69.775,177.313,17.289,152.226
C06862=1097.165,199.330,-69.752,177.309,17.289,152.227
C06863=1097.160,199.081,-69.729,177.306,17.290,152.228
C06864=1097.154,198.831,-69.705,177.302,17.289,152.228
C06865=1097.148,198.583,-69.681,177.299,17.289,152.229
C06866=1097.143,198.334,-69.658,177.295,17.289,152.229
C06867=1097.137,198.085,-69.634,177.292,17.289,152.230
C06868=1097.131,197.836,-69.611,177.288,17.289,152.231
C06869=1097.126,197.588,-69.587,177.285,17.289,152.231
C06870=1097.120,197.339,-69.564,177.282,17.289,152.232
C06871=1097.114,197.090,-69.541,177.278,17.289,152.233
C06872=1097.109,196.841,-69.517,177.275,17.288,152.233
C06873=1097.103,196.592,-69.493,177.271,17.288,152.234
C06874=1097.097,196.343,-69.470,177.268,17.289,152.235
C06875=1097.091,196.095,-69.447,177.265,17.288,152.235
C06876=1097.086,195.845,-69.423,177.261,17.288,152.236
C06877=1097.080,195.596,-69.400,177.258,17.288,152.237
C06878=1097.074,195.348,-69.377,177.254,17.288,152.237
C06879=1097.069,195.099,-69.353,177.251,17.288,152.238
C06880=1097.064,194.850,-69.330,177.248,17.288,152.238
C06881=1097.058,194.601,-69.307,177.244,17.288,152.239
C06882=1097.052,194.353,-69.283,177.242,17.288,152.240
C06883=1097.047,194.104,-69.260,177.238,17.288,152.240
C06884=1097.041,193.855,-69.237,177.235,17.288,152.241
C06885=1097.035,193.606,-69.214,177.231,17.288,152.242
C06886=1097.030,193.357,-69.191,177.228,17.287,152.242
C06887=1097.024,193.108,-69.167,177.225,17.288,152.243
C06888=1097.019,192.860,-69.144,177.221,17.287,152.244
C06889=1097.013,192.611,-69.121,177.218,17.287,152.244
C06890=1097.007,192.336,-69.095,177.214,17.287,152.245
C06891=1097.001,192.062,-69.070,177.211,17.287,152.245
C06892=1096.994,191.788,-69.044,177.207,17.286,152.246
C06893=1096.988,191.513,-69.019,177.203,17.287,152.247
C06894=1096.983,191.265,-68.996,177.200,17.287,152.248
C06895=1096.978,191.015,-68.973,177.196,17.286,152.248
C06896=1096.972,190.766,-68.950,177.193,17.286,152.249
C06897=1096.966,190.518,-68.927,177.190,17.286,152.249
C06898=1096.960,190.269,-68.904,177.186,17.286,152.250
C06899=1096.954,190.020,-68.880,177.183,17.286,152.251
C06900=1096.949,189.771,-68.856,177.180,17.286,152.251
C06901=1096.944,189.523,-68.834,177.177,17.286,152.252
C06902=1096.939,189.274,-68.811,177.174,17.286,152.253
C06903=1096.933,189.025,-68.788,177.170,17.285,152.253
C06904=1096.927,188.776,-68.765,177.167,17.285,152.254
C06905=1096.921,188.527,-68.742,177.164,17.285,152.254
C06906=1096.917,188.278,-68.719,177.160,17.285,152.255
C06907=1096.911,188.029,-68.696,177.157,17.285,152.256
C06908=1096.905,187.780,-68.673,177.153,17.284,152.256
C06909=1096.900,187.532,-68.651,177.150,17.285,152.257
C06910=1096.894,187.283,-68.628,177.147,17.284,152.257
C06911=1096.889,187.034,-68.605,177.143,17.284,152.258
C06912=1096.883,186.785,-68.582,177.141,17.284,152.259
C06913=1096.877,186.536,-68.559,177.137,17.284,152.259
C06914=1096.872,186.287,-68.535,177.134,17.284,152.260
C06915=1096.867,186.039,-68.513,177.131,17.283,152.260
C06916=1096.862,185.789,-68.491,177.127,17.283,152.261
C06917=1096.856,185.540,-68.468,177.124,17.283,152.262
C06918=1096.850,185.291,-68.445,177.121,17.283,152.262
C06919=1096.844,185.042,-68.422,177.117,17.283,152.263
C06920=1096.839,184.793,-68.399,177.114,17.283,152.263
C06921=1096.833,184.545,-68.376,177.111,17.283,152.264
C06922=1096.827,184.295,-68.354,177.107,17.282,152.265
C06923=1096.822,184.047,-68.332,177.105,17.283,152.265
C06924=1096.816,183.798,-68.309,177.101,17.283,152.266
C06925=1096.810,183.549,-68.286,177.098,17.282,152.267
C06926=1096.805,183.300,-68.264,177.095,17.282,152.267
C06927=1096.798,183.051,-68.241,177.091,17.282,152.268
C06928=1096.793,182.802,-68.218,177.088,17.282,152.268
C06929=1096.787,182.553,-68.195,177.085,17.282,152.269
C06930=1096.781,182.304,-68.173,177.081,17.282,152.270
C06931=1096.775,182.055,-68.151,177.079,17.282,152.270
C06932=1096.770,181.807,-68.128,177.075,17.282,152.271
C06933=1096.764,181.558,-68.106,177.072,17.282,152.272
C06934=1096.759,181.309,-68.083,177.069,17.281,152.272
C06935=1096.753,181.060,-68.060,177.065,17.281,152.273
C06936=1096.747,180.811,-68.038,177.062,17.281,152.273
C06937=1096.741,180.562,-68.016,177.059,17.281,152.274
C06938=1096.736,180.314,-67.993,177.055,17.280,152.275
C06939=1096.730,180.064,-67.971,177.053,17.281,152.275
C06940=1096.724,179.815,-67.948,177.049,17.281,152.276
C06941=1096.719,179.566,-67.926,177.046,17.280,152.276
C06942=1096.713,179.317,-67.903,177.043,17.281,152.277
C06943=1096.707,179.069,-67.881,177.039,17.280,152.278
C06944=1096.702,178.820,-67.859,177.036,17.280,152.278
C06945=1096.696,178.571,-67.836,177.033,17.280,152.279
C06946=1096.690,178.322,-67.814,177.029,17.280,152.279
C06947=1096.684,178.073,-67.791,177.027,17.280,152.280
C06948=1096.679,177.824,-67.770,177.024,17.280,152.281
C06949=1096.673,177.575,-67.747,177.020,17.280,152.281
C06950=1096.667,177.326,-67.725,177.017,17.279,152.282
C06951=1096.661,177.077,-67.702,177.014,17.279,152.282
C06952=1096.656,176.828,-67.681,177.010,17.279,152.283
C06953=1096.650,176.579,-67.658,177.007,17.279,152.284
C06954=1096.644,176.305,-67.633,177.003,17.278,152.284
C06955=1096.638,176.030,-67.609,177.000,17.278,152.285
C06956=1096.631,175.755,-67.584,176.997,17.278,152.285
C06957=1096.625,175.480,-67.560,176.993,17.278,152.286
C06958=1096.620,175.231,-67.537,176.990,17.278,152.287
C06959=1096.614,174.983,-67.516,176.987,17.278,152.287
C06960=1096.609,174.733,-67.493,176.983,17.277,152.288
C06961=1096.602,174.485,-67.471,176.980,17.277,152.288
C06962=1096.597,174.236,-67.449,176.977,17.278,152.289
C06963=1096.592,173.987,-67.427,176.974,17.277,152.290
C06964=1096.586,173.738,-67.405,176.971,17.277,152.290
C06965=1096.581,173.489,-67.383,176.968,17.277,152.291
C06966=1096.575,173.240,-67.361,176.964,17.276,152.291
C06967=1096.569,172.991,-67.338,176.961,17.276,152.292
C06968=1096.564,172.742,-67.316,176.958,17.275,152.292
C06969=1096.558,172.493,-67.295,176.955,17.276,152.293
C06970=1096.552,172.243,-67.272,176.952,17.275,152.294
C06971=1096.547,171.996,-67.250,176.949,17.276,152.294
C06972=1096.541,171.746,-67.228,176.945,17.275,152.295
C06973=1096.536,171.498,-67.207,176.942,17.275,152.295
C06974=1096.530,171.248,-67.185,176.939,17.274,152.296
C06975=1096.525,170.999,-67.163,176.936,17.274,152.297
C06976=1096.519,170.751,-67.141,176.933,17.274,152.297
C06977=1096.513,170.501,-67.118,176.930,17.274,152.298
C06978=1096.508,170.253,-67.097,176.927,17.274,152.298
C06979=1096.502,170.003,-67.075,176.923,17.273,152.299
C06980=1096.497,169.755,-67.054,176.920,17.273,152.299
C06981=1096.491,169.505,-67.031,176.917,17.273,152.300
C06982=1096.485,169.257,-67.009,176.914,17.273,152.300
C06983=1096.480,169.008,-66.987,176.911,17.273,152.301
C06984=1096.474,168.759,-66.965,176.908,17.272,152.302
C06985=1096.469,168.510,-66.944,176.905,17.272,152.302
C06986=1096.463,168.260,-66.922,176.901,17.272,152.303
C06987=1096.458,168.012,-66.900,176.898,17.271,152.303
C06988=1096.452,167.762,-66.878,176.896,17.271,152.304
C06989=1096.447,167.514,-66.857,176.892,17.271,152.304
C06990=1096.441,167.264,-66.835,176.890,17.270,152.305
C06991=1096.436,167.016,-66.813,176.886,17.270,152.305
C06992=1096.430,166.766,-66.791,176.883,17.270,152.306
C06993=1096.425,166.518,-66.770,176.880,17.269,152.306
C06994=1096.419,166.268,-66.748,176.877,17.270,152.307
C06995=1096.414,166.020,-66.726,176.874,17.269,152.308
C06996=1096.408,165.770,-66.704,176.871,17.269,152.308
C06997=1096.403,165.522,-66.683,176.868,17.269,152.309
C06998=1096.397,165.272,-66.661,176.864,17.268,152.309
C06999=1096.392,165.024,-66.640,176.862,17.268,152.310
C07000=1096.386,164.774,-66.617,176.859,17.268,152.310
C07001=1096.381,164.526,-66.596,176.856,17.267,152.311
C07002=1096.375,164.276,-66.574,176.852,17.267,152.311
C07003=1096.370,164.028,-66.553,176.849,17.267,152.312
C07004=1096.365,163.779,-66.531,176.846,17.266,152.312
C07005=1096.359,163.530,-66.509,176.844,17.266,152.313
C07006=1096.353,163.281,-66.489,176.840,17.266,152.313
C07007=1096.348,163.031,-66.466,176.837,17.265,152.314
C07008=1096.342,162.783,-66.445,176.834,17.265,152.314
C07009=1096.337,162.534,-66.423,176.831,17.264,152.315
C07010=1096.331,162.285,-66.402,176.828,17.265,152.315
C07011=1096.326,162.036,-66.380,176.825,17.264,152.316
C07012=1096.321,161.786,-66.359,176.822,17.264,152.317
C07013=1096.315,161.537,-66.338,176.819,17.263,152.317
C07014=1096.309,161.288,-66.316,176.816,17.263,152.318
C07015=1096.303,161.040,-66.295,176.812,17.262,152.318
C07016=1096.299,160.790,-66.274,176.810,17.263,152.319
C07017=1096.293,160.541,-66.252,176.807,17.262,152.319
C07018=1096.286,160.266,-66.229,176.803,17.262,152.320
C07019=1096.280,159.992,-66.205,176.800,17.262,152.320
C07020=1096.274,159.717,-66.182,176.797,17.261,152.321
C07021=1096.268,159.442,-66.158,176.794,17.261,152.321
C07022=1096.262,159.192,-66.136,176.790,17.261,152.322
C07023=1096.257,158.943,-66.116,176.787,17.260,152.323
C07024=1096.250,158.694,-66.094,176.784,17.260,152.323
C07025=1096.245,158.445,-66.073,176.781,17.260,152.324
C07026=1096.240,158.196,-66.052,176.779,17.260,152.324
C07027=1096.233,157.947,-66.030,176.775,17.259,152.325
C07028=1096.228,157.699,-66.009,176.772,17.259,152.325
C07029=1096.223,157.448,-65.988,176.769,17.259,152.326
C07030=1096.217,157.200,-65.966,176.766,17.258,152.326
C07031=1096.212,156.952,-65.945,176.763,17.258,152.327
C07032=1096.206,156.702,-65.924,176.760,17.258,152.327
C07033=1096.200,156.453,-65.903,176.757,17.257,152.328
C07034=1096.195,156.204,-65.882,176.754,17.257,152.328
C07035=1096.189,155.955,-65.861,176.751,17.257,152.329
C07036=1096.183,155.706,-65.839,176.748,17.256,152.329
C07037=1096.178,155.457,-65.819,176.745,17.256,152.330
C07038=1096.172,155.208,-65.797,176.742,17.255,152.330
C07039=1096.167,154.959,-65.777,176.739,17.255,152.331
C07040=1096.160,154.710,-65.755,176.736,17.255,152.331
C07041=1096.155,154.461,-65.735,176.733,17.255,152.332
C07042=1096.150,154.212,-65.713,176.730,17.254,152.332
C07043=1096.144,153.962,-65.692,176.727,17.254,152.333
C07044=1096.138,153.714,-65.671,176.725,17.254,152.333
C07045=1096.133,153.465,-65.650,176.721,17.253,152.334
C07046=1096.127,153.215,-65.629,176.718,17.253,152.334
C07047=1096.121,152.966,-65.608,176.715,17.252,152.335
C07048=1096.116,152.717,-65.588,176.712,17.252,152.336
C07049=1096.111,152.469,-65.566,176.710,17.252,152.336
C07050=1096.105,152.219,-65.546,176.706,17.251,152.336
C07051=1096.099,151.970,-65.524,176.703,17.251,152.337
C07052=1096.094,151.721,-65.504,176.700,17.250,152.337
C07053=1096.088,151.471,-65.483,176.698,17.251,152.338
C07054=1096.083,151.223,-65.462,176.695,17.250,152.338
C07055=1096.077,150.974,-65.442,176.691,17.249,152.339
C07056=1096.071,150.726,-65.420,176.688,17.249,152.340
C07057=1096.065,150.476,-65.399,176.686,17.249,152.340
C07058=1096.060,150.227,-65.379,176.683,17.249,152.341
C07059=1096.054,149.978,-65.358,176.680,17.248,152.341
C07060=1096.048,149.728,-65.337,176.676,17.247,152.342
C07061=1096.043,149.479,-65.316,176.674,17.247,152.342
C07062=1096.038,149.230,-65.296,176.671,17.247,152.342
C07063=1096.032,148.982,-65.275,176.668,17.247,152.343
C07064=1096.026,148.733,-65.254,176.665,17.246,152.343
C07065=1096.021,148.483,-65.233,176.662,17.246,152.344
C07066=1096.015,148.234,-65.213,176.659,17.245,152.344
C07067=1096.010,147.985,-65.192,176.656,17.245,152.345
C07068=1096.004,147.736,-65.172,176.653,17.244,152.345
C07069=1095.998,147.487,-65.151,176.650,17.244,152.346
C07070=1095.993,147.237,-65.130,176.648,17.244,152.346
C07071=1095.987,146.989,-65.109,176.644,17.243,152.347
C07072=1095.981,146.740,-65.089,176.641,17.243,152.347
C07073=1095.975,146.490,-65.068,176.639,17.243,152.348
C07074=1095.970,146.241,-65.047,176.636,17.242,152.348
C07075=1095.965,145.992,-65.027,176.633,17.242,152.349
C07076=1095.959,145.743,-65.007,176.630,17.241,152.349
C07077=1095.953,145.495,-64.986,176.627,17.241,152.350
C07078=1095.947,145.245,-64.965,176.624,17.240,152.350
C07079=1095.941,144.996,-64.945,176.621,17.240,152.351
C07080=1095.936,144.747,-64.924,176.618,17.239,152.351
C07081=1095.931,144.498,-64.904,176.616,17.240,152.352
C07082=1095.925,144.222,-64.881,176.613,17.239,152.352
C07083=1095.918,143.948,-64.859,176.609,17.239,152.353
C07084=1095.912,143.672,-64.836,176.606,17.238,152.353
C07085=1095.906,143.396,-64.814,176.602,17.237,152.354
C07086=1095.900,143.148,-64.792,176.600,17.237,152.354
C07087=1095.894,142.899,-64.772,176.597,17.236,152.355
C07088=1095.889,142.650,-64.752,176.594,17.236,152.355
C07089=1095.883,142.400,-64.731,176.591,17.236,152.356
C07090=1095.877,142.151,-64.711,176.589,17.235,152.356
C07091=1095.872,141.902,-64.690,176.585,17.235,152.357
C07092=1095.866,141.653,-64.670,176.582,17.234,152.357
C07093=1095.861,141.404,-64.650,176.580,17.234,152.357
C07094=1095.856,141.154,-64.630,176.577,17.233,152.358
C07095=1095.850,140.906,-64.610,176.574,17.233,152.358
C07096=1095.844,140.657,-64.589,176.571,17.232,152.359
C07097=1095.839,140.407,-64.569,176.568,17.232,152.359
C07098=1095.833,140.158,-64.549,176.565,17.231,152.360
C07099=1095.827,139.909,-64.528,176.562,17.231,152.360
C07100=1095.821,139.660,-64.508,176.560,17.231,152.361
C07101=1095.816,139.411,-64.487,176.557,17.230,152.361
C07102=1095.810,139.162,-64.468,176.554,17.229,152.362
C07103=1095.805,138.913,-64.447,176.551,17.229,152.362
C07104=1095.799,138.664,-64.427,176.549,17.229,152.363
C07105=1095.794,138.414,-64.407,176.546,17.228,152.363
C07106=1095.788,138.166,-64.387,176.543,17.227,152.363
C07107=1095.783,137.916,-64.367,176.540,17.228,152.364
C07108=1095.777,137.668,-64.347,176.537,17.227,152.364
C07109=1095.771,137.418,-64.326,176.534,17.226,152.365
C07110=1095.765,137.168,-64.307,176.531,17.226,152.365
C07111=1095.760,136.919,-64.286,176.529,17.225,152.366
C07112=1095.754,136.670,-64.266,176.526,17.225,152.366
C07113=1095.748,136.422,-64.246,176.523,17.224,152.367
C07114=1095.743,136.172,-64.226,176.520,17.224,152.367
C07115=1095.737,135.923,-64.206,176.517,17.223,152.368
C07116=1095.732,135.674,-64.186,176.514,17.223,152.368
C07117=1095.726,135.425,-64.166,176.511,17.222,152.368
C07118=1095.720,135.176,-64.145,176.509,17.222,152.369
C07119=1095.715,134.927,-64.126,176.506,17.221,152.369
C07120=1095.709,134.678,-64.106,176.503,17.221,152.370
C07121=1095.704,134.429,-64.085,176.501,17.220,152.370
C07122=1095.698,134.179,-64.066,176.498,17.220,152.371
C07123=1095.693,133.930,-64.046,176.495,17.219,152.371
C07124=1095.687,133.681,-64.026,176.492,17.219,152.372
C07125=1095.681,133.432,-64.006,176.489,17.218,152.372
C07126=1095.676,133.183,-63.986,176.486,17.218,152.372
C07127=1095.670,132.934,-63.966,176.483,17.217,152.373
C07128=1095.664,132.684,-63.947,176.481,17.217,152.373
C07129=1095.659,132.435,-63.926,176.478,17.216,152.374
C07130=1095.653,132.186,-63.907,176.475,17.215,152.374
C07131=1095.647,131.937,-63.887,176.473,17.215,152.375
C07132=1095.642,131.688,-63.866,176.470,17.215,152.375
C07133=1095.636,131.439,-63.847,176.467,17.214,152.375
C07134=1095.630,131.190,-63.827,176.465,17.214,152.376
C07135=1095.624,130.940,-63.808,176.462,17.213,152.376
C07136=1095.618,130.691,-63.788,176.458,17.213,152.377
C07137=1095.613,130.442,-63.768,176.456,17.212,152.377
C07138=1095.607,130.193,-63.748,176.453,17.212,152.378
C07139=1095.602,129.943,-63.729,176.450,17.211,152.378
C07140=1095.596,129.695,-63.709,176.447,17.210,152.378
C07141=1095.590,129.445,-63.690,176.445,17.210,152.379
C07142=1095.584,129.196,-63.670,176.442,17.209,152.379
C07143=1095.579,128.947,-63.650,176.439,17.208,152.380
C07144=1095.573,128.698,-63.630,176.437,17.209,152.380
C07145=1095.567,128.448,-63.611,176.434,17.208,152.381
C07146=1095.561,128.174,-63.589,176.431,17.207,152.381
C07147=1095.555,127.899,-63.567,176.428,17.206,152.381
C07148=1095.548,127.623,-63.546,176.424,17.206,152.382
C07149=1095.542,127.347,-63.524,176.422,17.205,152.382
C07150=1095.537,127.098,-63.505,176.419,17.205,152.383
C07151=1095.531,126.849,-63.485,176.416,17.204,152.383
C07152=1095.526,126.600,-63.465,176.413,17.203,152.384
C07153=1095.520,126.351,-63.446,176.411,17.203,152.384
C07154=1095.514,126.102,-63.426,176.408,17.203,152.384
C07155=1095.508,125.852,-63.407,176.405,17.202,152.385
C07156=1095.502,125.604,-63.387,176.403,17.202,152.385
C07157=1095.496,125.354,-63.368,176.400,17.201,152.386
C07158=1095.492,125.104,-63.348,176.397,17.200,152.386
C07159=1095.486,124.855,-63.329,176.395,17.200,152.387
C07160=1095.480,124.607,-63.309,176.392,17.199,152.387
C07161=1095.475,124.357,-63.290,176.389,17.198,152.387
C07162=1095.469,124.108,-63.271,176.387,17.198,152.388
C07163=1095.463,123.859,-63.251,176.384,17.197,152.388
C07164=1095.457,123.610,-63.231,176.381,17.197,152.389
C07165=1095.452,123.360,-63.212,176.379,17.196,152.389
C07166=1095.446,123.111,-63.193,176.376,17.195,152.389
C07167=1095.441,122.863,-63.173,176.373,17.194,152.390
C07168=1095.435,122.613,-63.154,176.371,17.194,152.390
C07169=1095.429,122.364,-63.135,176.368,17.193,152.390
C07170=1095.424,122.114,-63.116,176.365,17.193,152.391
C07171=1095.418,121.865,-63.096,176.363,17.192,152.391
C07172=1095.412,121.617,-63.077,176.360,17.192,152.392
C07173=1095.407,121.367,-63.058,176.357,17.191,152.392
C07174=1095.401,121.118,-63.038,176.355,17.190,152.392
C07175=1095.395,120.869,-63.019,176.352,17.190,152.393
C07176=1095.390,120.619,-63.000,176.349,17.189,152.393
C07177=1095.385,120.370,-62.981,176.347,17.189,152.394
C07178=1095.379,120.122,-62.961,176.344,17.188,152.394
C07179=1095.373,119.872,-62.942,176.341,17.187,152.394
C07180=1095.367,119.623,-62.923,176.339,17.186,152.395
C07181=1095.362,119.374,-62.904,176.336,17.186,152.395
C07182=1095.356,119.125,-62.884,176.333,17.185,152.396
C07183=1095.351,118.875,-62.865,176.331,17.185,152.396
C07184=1095.345,118.626,-62.846,176.328,17.183,152.396
C07185=1095.340,118.377,-62.827,176.325,17.183,152.397
C07186=1095.334,118.128,-62.808,176.323,17.182,152.397
C07187=1095.329,117.878,-62.789,176.320,17.182,152.397
C07188=1095.323,117.629,-62.769,176.317,17.180,152.398
C07189=1095.318,117.380,-62.750,176.315,17.180,152.398
C07190=1095.312,117.131,-62.731,176.312,17.180,152.399
C07191=1095.306,116.881,-62.712,176.309,17.179,152.399
C07192=1095.301,116.632,-62.693,176.307,17.178,152.399
C07193=1095.296,116.383,-62.674,176.304,17.177,152.400
C07194=1095.290,116.133,-62.655,176.302,17.177,152.400
C07195=1095.285,115.885,-62.636,176.299,17.176,152.400
C07196=1095.279,115.635,-62.616,176.296,17.175,152.401
C07197=1095.274,115.386,-62.597,176.294,17.175,152.401
C07198=1095.268,115.137,-62.578,176.291,17.174,152.401
C07199=1095.263,114.888,-62.559,176.288,17.173,152.402
C07200=1095.256,114.639,-62.540,176.286,17.172,152.402
C07201=1095.251,114.390,-62.522,176.283,17.172,152.402
C07202=1095.246,114.140,-62.502,176.280,17.171,152.403
C07203=1095.240,113.890,-62.484,176.278,17.171,152.403
C07204=1095.235,113.642,-62.465,176.275,17.169,152.404
C07205=1095.229,113.393,-62.446,176.273,17.169,152.404
C07206=1095.223,113.143,-62.427,176.270,17.168,152.404
C07207=1095.217,112.894,-62.408,176.268,17.167,152.405
C07208=1095.212,112.645,-62.389,176.265,17.167,152.405
C07209=1095.206,112.396,-62.370,176.262,17.166,152.405
C07210=1095.200,112.121,-62.349,176.260,17.165,152.406
C07211=1095.194,111.845,-62.328,176.257,17.164,152.406
C07212=1095.188,111.569,-62.307,176.254,17.163,152.407
C07213=1095.182,111.294,-62.288,176.251,17.163,152.407
C07214=1095.176,111.045,-62.269,176.249,17.162,152.407
C07215=1095.169,110.795,-62.250,176.246,17.161,152.408
C07216=1095.164,110.547,-62.231,176.244,17.161,152.408
C07217=1095.159,110.297,-62.212,176.241,17.160,152.408
C07218=1095.153,110.047,-62.194,176.238,17.159,152.409
C07219=1095.147,109.799,-62.175,176.236,17.159,152.409
C07220=1095.142,109.549,-62.156,176.233,17.158,152.409
C07221=1095.136,109.300,-62.138,176.230,17.157,152.410
C07222=1095.131,109.051,-62.119,176.228,17.156,152.410
C07223=1095.124,108.802,-62.100,176.225,17.156,152.410
C07224=1095.118,108.552,-62.081,176.223,17.155,152.411
C07225=1095.114,108.303,-62.063,176.220,17.154,152.411
C07226=1095.107,108.054,-62.044,176.217,17.153,152.412
C07227=1095.102,107.805,-62.025,176.215,17.153,152.412
C07228=1095.096,107.555,-62.007,176.212,17.152,152.412
C07229=1095.090,107.306,-61.988,176.211,17.151,152.412
C07230=1095.086,107.057,-61.970,176.208,17.151,152.413
C07231=1095.079,106.807,-61.951,176.205,17.149,152.413
C07232=1095.074,106.559,-61.933,176.203,17.149,152.414
C07233=1095.068,106.309,-61.915,176.200,17.148,152.414
C07234=1095.062,106.060,-61.895,176.197,17.147,152.414
C07235=1095.057,105.810,-61.878,176.195,17.146,152.415
C07236=1095.051,105.561,-61.859,176.192,17.146,152.415
C07237=1095.045,105.313,-61.840,176.190,17.145,152.415
C07238=1095.040,105.063,-61.822,176.187,17.144,152.416
C07239=1095.035,104.814,-61.803,176.185,17.143,152.416
C07240=1095.029,104.564,-61.785,176.182,17.143,152.416
C07241=1095.024,104.315,-61.766,176.180,17.142,152.417
C07242=1095.017,104.066,-61.748,176.177,17.141,152.417
C07243=1095.012,103.817,-61.729,176.175,17.140,152.417
C07244=1095.006,103.567,-61.711,176.172,17.139,152.418
C07245=1095.001,103.318,-61.692,176.170,17.139,152.418
C07246=1094.995,103.069,-61.675,176.167,17.138,152.418
C07247=1094.990,102.820,-61.656,176.165,17.137,152.419
C07248=1094.984,102.570,-61.638,176.162,17.136,152.419
C07249=1094.979,102.322,-61.619,176.160,17.135,152.419
C07250=1094.973,102.072,-61.601,176.157,17.135,152.419
C07251=1094.968,101.822,-61.583,176.155,17.134,152.420
C07252=1094.961,101.573,-61.564,176.153,17.133,152.420
C07253=1094.957,101.324,-61.546,176.150,17.132,152.420
C07254=1094.950,101.075,-61.527,176.147,17.131,152.421
C07255=1094.945,100.826,-61.510,176.145,17.131,152.421
C07256=1094.939,100.576,-61.490,176.142,17.129,152.421
